// Wsuń/zamknij
bClose_Cmd R= ( (stDigInOut.bI_Closed OR fbTON_CloseTimer.Q) AND NOT bI_SusteinClosePos) OR NOT bI_Control_Ready;
//bClose_Cmd R= ( (bI_Closed OR (fbTON_CloseTimer.Q AND FALSE)) AND NOT bI_SusteinClosePos) OR NOT bI_Control_Ready;
stDigInOut.bQ_Close := bClose_Cmd AND (SEL(bI_MANUAL_CMD, NOT bI_CloseInterlock, NOT (bI_CloseInterlock AND bI_RespectInterlockInMAN)) OR bQ_Closed);
stDigInOut.bQ_Open R= stDigInOut.bQ_Close;

// Wysuń/otwórz
bOpen_Cmd R= ( (stDigInOut.bI_Opened OR fbTON_OpenTimer.Q) AND NOT bI_SusteinOpenPos) OR NOT bI_Control_Ready;
//bOpen_Cmd R= ( (bI_Opened OR (fbTON_OpenTimer.Q AND FALSE)) AND NOT bI_SusteinOpenPos) OR NOT bI_Control_Ready;
stDigInOut.bQ_Open := bOpen_Cmd AND (SEL(bI_MANUAL_CMD, NOT bI_OpenInterlock, NOT (bI_OpenInterlock AND bI_RespectInterlockInMAN)) OR bQ_Opened);
stDigInOut.bQ_Close R= stDigInOut.bQ_Open;

// Określenie sygnałów zamknięcia/otwarcia
fbFTrig_Opened (CLK := stDigInOut.bI_Opened);
fbFTrig_Closed (CLK := stDigInOut.bI_Closed);
IF bAllowOverCrossPosition THEN
	bQ_Opened R= (NOT stDigInOut.bQ_Open AND fbFTrig_Opened.Q) OR stDigInOut.bI_Closed; 
	bQ_Closed R= (NOT stDigInOut.bQ_Close AND fbFTrig_Closed.Q) OR stDigInOut.bI_Opened;
	bQ_Opened S= stDigInOut.bI_Opened;
	bQ_Closed S= stDigInOut.bI_Closed;
ELSE
	bQ_Opened := stDigInOut.bI_Opened;
	bQ_Closed := stDigInOut.bI_Closed; 
END_IF
bCmdActive := FALSE;

// Kontrola czasu pracy siłownika
IF fbTON_OpenTimer.IN AND NOT (stDigInOut.bQ_Open AND NOT bQ_Opened) AND NOT fbTON_OpenTimer.Q THEN
	fMeanFilter(rInputValue := TIME_TO_REAL(fbTON_OpenTimer.ET), rDelta := 10.0, rMeanValue := rOpenMeanTime);
END_IF
fbTON_OpenTimer(IN := stDigInOut.bQ_Open AND NOT bQ_Opened, PT:= REAL_TO_TIME(1000.0*rI_OpenTime));

IF fbTON_CloseTimer.IN AND NOT (stDigInOut.bQ_Close AND NOT bQ_Closed) AND NOT fbTON_CloseTimer.Q THEN
	fMeanFilter(rInputValue := TIME_TO_REAL(fbTON_CloseTimer.ET), rDelta := 10.0, rMeanValue := rCloseMeanTime);
END_IF
fbTON_CloseTimer(IN := stDigInOut.bQ_Close AND NOT bQ_Closed, PT:= REAL_TO_TIME(1000.0*rI_CloseTime));

bInMovement:= fbTON_OpenTimer.IN OR fbTON_CloseTimer.IN;

// Kontrola błędów w pracy
fbTON_controlReady(IN:= bI_Control_Ready, PT:= T#5S);		// Alarmuj tylko po powrocie sygnału gotowości napędów

// Błąd osiągnięcia pozycji otwórz w odpowiednim czasie
IF fbTON_OpenTimer.Q AND fbTON_controlReady.Q AND __ISVALIDREF(fbAlarmTab) THEN
	IF NOT bOpenTimeExceedAlSend THEN
		fbAlarmTab.mPushRow(nAlarmClass:= enAlarmClasses.Error, sMachineId := sActuatorId, sEventDesc := 'Open time exceeded, open position not achieved', dwErrorId := 0);
		bOpenTimeExceedAlSend := TRUE;
	END_IF
ELSE
	bOpenTimeExceedAlSend := FALSE;
END_IF

// Błąd osiągnięcia pozycji zamknij w odpowiednim czasie
IF fbTON_CloseTimer.Q AND fbTON_controlReady.Q AND __ISVALIDREF(fbAlarmTab) THEN
	IF NOT bCloseTimeExceedAlSend THEN
		fbAlarmTab.mPushRow(nAlarmClass:= enAlarmClasses.Error, sMachineId := sActuatorId, sEventDesc := 'Close time exceeded, close position not achieved', dwErrorId := 0);
		bCloseTimeExceedAlSend := TRUE;
	END_IF
ELSE
	bCloseTimeExceedAlSend := FALSE;
END_IF

// Utracenie pozycji otwarcia
fbFTRIG_OpenPosition(CLK:= bQ_Opened);
IF fbFTRIG_OpenPosition.Q AND NOT stDigInOut.bQ_Open AND NOT stDigInOut.bQ_Close AND fbTON_controlReady.Q AND bEnPossLossAlarm AND __ISVALIDREF(fbAlarmTab) THEN
	fbAlarmTab.mPushRow(nAlarmClass:= enAlarmClasses.Error, sMachineId := sActuatorId, sEventDesc := 'Loss open position', dwErrorId := 0);
END_IF

// Utracenie pozycji zamknięcia
fbFTRIG_ClosePosition(CLK:= bQ_Closed);
IF fbFTRIG_ClosePosition.Q AND NOT stDigInOut.bQ_Open AND NOT stDigInOut.bQ_Close AND fbTON_controlReady.Q AND bEnPossLossAlarm AND __ISVALIDREF(fbAlarmTab) THEN
	fbAlarmTab.mPushRow(nAlarmClass:= enAlarmClasses.Error, sMachineId := sActuatorId, sEventDesc := 'Loss close position', dwErrorId := 0);
END_IF

// Kontrola pracy krańcówek
fbRTrig_Open(CLK := stDigInOut.bI_Opened);
fbRTrig_Close(CLK := stDigInOut.bI_Closed);

IF ((stDigInOut.bQ_Open AND fbRTrig_Close.Q AND NOT bAllowOverCrossPosition) OR (stDigInOut.bQ_Close AND fbRTrig_Open.Q AND NOT bAllowOverCrossPosition) OR (stDigInOut.bI_Opened AND stDigInOut.bI_Closed) AND fbTON_controlReady.Q ) AND __ISVALIDREF(fbAlarmTab) THEN
	IF NOT bSwitchesErrorAlSend THEN
		fbAlarmTab.mPushRow(nAlarmClass:= enAlarmClasses.Error, sMachineId := sActuatorId, sEventDesc := 'End stops error', dwErrorId := 0);
	END_IF
ELSE
	bSwitchesErrorAlSend := FALSE;
END_IF

// Ilość cykli pracy
fbRTrig_Ctr_Open (CLK := stDigInOut.bQ_Open);
fbRTrig_Ctr_Close (CLK := stDigInOut.bQ_Close);
IF fbRTrig_Ctr_Open.Q OR fbRTrig_Ctr_Close.Q THEN
	diNbOfOperations := diNbOfOperations+1;
END_IF

ACTION ACT_Stop:
stDigInOut.bQ_Open := stDigInOut.bQ_Close := FALSE;
END_ACTION

METHOD mClose : BOOL
VAR_INPUT
	bManCtrl:BOOL;
END_VAR
IF bManCtrl THEN
	bClose_Cmd S= bI_MANUAL_CMD;
ELSE
	bClose_Cmd S= NOT bI_MANUAL_CMD;
END_IF
bOpen_Cmd R= bClose_Cmd;
bCmdActive := TRUE;
(*bResult := bClose_Cmd;
IF bManCtrl THEN
	bClose_Cmd S= bI_MANUAL_CMD AND NOT (bI_CloseInterlock AND bI_RespectInterlockInMAN);
ELSE
	bClose_Cmd S= NOT bI_MANUAL_CMD AND NOT bI_CloseInterlock;
END_IF
*)
END_METHOD

METHOD mOpen : BOOL
VAR_INPUT
	bManCtrl:BOOL;
END_VAR
IF bManCtrl THEN
	bOpen_Cmd := bI_MANUAL_CMD;
ELSE
	bOpen_Cmd := NOT bI_MANUAL_CMD;
END_IF
bClose_Cmd R= bOpen_Cmd;
bCmdActive := TRUE;
//bResult := bClose_Cmd;
END_METHOD

METHOD mReset : BOOL
VAR_INPUT
END_VAR
// Reset błędów 
fbTON_OpenTimer(IN:= FALSE);
fbTON_CloseTimer(IN:= FALSE);
END_METHOD

METHOD mStop : BOOL
VAR_INPUT
	bManCtrl:BOOL;
END_VAR
IF bManCtrl AND bI_MANUAL_CMD THEN
	bOpen_Cmd := bClose_Cmd := FALSE;
	ACT_Stop();
END_IF
bCmdActive := TRUE;
END_METHOD

END_FUNCTION_BLOCK

// Common/Actuator/fbActuatorV2
FUNCTION_BLOCK fbActuatorV2
VAR_IN_OUT
	
END_VAR
VAR_INPUT
	bControl_Rdy			:BOOL;		// Sygnał gotowości sterowania, sygnały otwórz/zamknij ustawiane tylko gdy jest gotowość
	bInterlock_Open			:BOOL;		// Sygnał blokady otwierania zaworu/napędu (kolizja z innymi elementami)
	bInterlock_Close		:BOOL;		// Sygnał blokady zamykania zaworu/napędu (kolizja z innymi elementami)
	bSusteinOutput			:BOOL;		// Po dojściu do pozycji zadanej podtrzymaj sygnał sterujący - stosować np. dla zaworów 5/2 w celu podtrzymania położenia
	bAllowOvercrossingPos	:BOOL;		// Ustawiaj sygnał otwórz/zamknij gdy ustawi się odpowiednia krańcówka oraz gdy aktywny sygnał sterujący (zejście z krańcówki przy podtrzymaniu nie powoduje zaniku sygnału otwarcia/zamknięcia)
	rOpenTime				:REAL;		//
	rCloseTime				:REAL;
END_VAR
VAR
	stInOuts: stActuatorInOuts;
	fbTON_AllowToNextOper	:TON;
	fbFTrig_Opened: F_TRIG;
	fbFTrig_Closed: F_TRIG;	
	bOpenPos_Overcrossed: BOOL;
	bClosePos_Overcrossed: BOOL;
	fbRTrig_Ctr_OPEN, fbRTrig_Ctr_CLOSE: R_TRIG;
	fbTON_ResetSustein: TON;
END_VAR

VAR PERSISTENT
	udiNbOfOperations:UDINT;
END_VAR

// Reset sygnałów sterujących po osiągnięciu pozycji
fbTON_ResetSustein(IN:= (stInOuts.bQ_Open AND Opened AND NOT bSusteinOutput) OR (stInOuts.bQ_Close AND Closed AND NOT bSusteinOutput),PT:= T#250MS);
stInOuts.bQ_Open R= stInOuts.bQ_Open AND ( (bInterlock_Open AND NOT Opened) OR fbTON_ResetSustein.Q);
stInOuts.bQ_Close R= stInOuts.bQ_Close AND ( (bInterlock_Close AND NOT Closed) OR fbTON_ResetSustein.Q);

// Zezwolenie na kolejną operację nie szybciej niż co 50 ms
fbTON_AllowToNextOper(IN:= NOT stInOuts.bQ_Open AND NOT stInOuts.bQ_Close, PT:= T#50MS);

// Określenie sygnałów zamknięcia/otwarcia
fbFTrig_Opened (CLK := stInOuts.bI_Opened);
fbFTrig_Closed (CLK := stInOuts.bI_Closed);
bOpenPos_Overcrossed S= stInOuts.bQ_Open AND fbFTrig_Opened.Q;
bOpenPos_Overcrossed R= stInOuts.bQ_Close AND fbFTrig_Opened.Q;
bClosePos_Overcrossed S= stInOuts.bQ_Close AND fbFTrig_Closed.Q;
bClosePos_Overcrossed R= stInOuts.bQ_Open AND fbFTrig_Closed.Q;

// Ilość cykli pracy
fbRTrig_Ctr_OPEN (CLK := stInOuts.bQ_Open);
fbRTrig_Ctr_CLOSE (CLK := stInOuts.bQ_Close);
IF fbRTrig_Ctr_OPEN.Q OR fbRTrig_Ctr_CLOSE.Q THEN
	udiNbOfOperations := udiNbOfOperations+1;
END_IF

METHOD mClose : BOOL
IF Closed THEN		// Siłownik zamknięty spróbuj ustawić wyjście		
	stInOuts.bQ_Open := FALSE;
	stInOuts.bQ_Close S= bControl_Rdy AND bSusteinOutput; 
	mClose := TRUE;
ELSE	// Jeśli siłownik nie zamknięty spróbuj ustawić wyjscie
	stInOuts.bQ_Close S= stInOuts.bQ_Open R= NOT bInterlock_Close AND bControl_Rdy;
END_IF
END_METHOD

METHOD mOpen : BOOL
IF Opened THEN			// Siłownik otwarty spróbuj ustawić wyjście	
	stInOuts.bQ_Close := FALSE;
	stInOuts.bQ_Open S= bControl_Rdy AND bSusteinOutput; 
	mOpen := TRUE;
ELSE					// Jeśli siłownik nie zamknięty spróbuj ustawić wyjscie
	stInOuts.bQ_Open S= stInOuts.bQ_Close R= NOT bInterlock_Open AND bControl_Rdy;
END_IF
END_METHOD

METHOD mReset : BOOL
END_METHOD

METHOD mStop : BOOL
stInOuts.bQ_Open := stInOuts.bQ_Close := FALSE;
END_METHOD

PROPERTY Closed : BOOL
GET
Closed := stInOuts.bI_Closed OR (bAllowOvercrossingPos AND bClosePos_Overcrossed);
END_GET
END_PROPERTY

PROPERTY CmdsCounter : UDINT
GET
CmdsCounter := udiNbOfOperations;
END_GET
SET
udiNbOfOperations := CmdsCounter;
END_SET
END_PROPERTY

PROPERTY Moving : BOOL
GET
Moving := (stInOuts.bQ_Open AND NOT Opened)OR (stInOuts.bQ_Close AND NOT Closed);
END_GET
END_PROPERTY

PROPERTY Opened : BOOL
GET
Opened := stInOuts.bI_Opened OR (bAllowOvercrossingPos AND bOpenPos_Overcrossed);
END_GET
END_PROPERTY

END_FUNCTION_BLOCK

// Common/AlarmTable/f_AlarmClassToUINT
FUNCTION f_AlarmClassToUINT : UINT
VAR_INPUT
	nAlarmType:enAlarmClasses;
END_VAR
VAR
END_VAR

CASE nAlarmType OF
	enAlarmClasses.None, enAlarmClasses.Info:
		f_AlarmClassToUINT:= 1;
	enAlarmClasses.Warning:
		f_AlarmClassToUINT:= 2;
	enAlarmClasses.Error:
		f_AlarmClassToUINT:= 3;
	enAlarmClasses.Quality:
		f_AlarmClassToUINT:= 4;
	enAlarmClasses.Maintenance:
		f_AlarmClassToUINT:= 5;
	enAlarmClasses.IT:
		f_AlarmClassToUINT:= 6;
	enAlarmClasses.Developer:
		f_AlarmClassToUINT:= 7;
END_CASE

END_FUNCTION

// Common/AlarmTable/f_AlarmEnableTest
FUNCTION f_AlarmEnableTest : BOOL
VAR_INPUT
	uiLogSettings:UINT;
	nAlarmType:enAlarmClasses;
END_VAR
VAR
	iBase:UINT := 1;
	uiBitNb: UINT;
END_VAR

CASE nAlarmType OF
	enAlarmClasses.None:
		f_AlarmEnableTest := FALSE;
		RETURN;	
	enAlarmClasses.Info:
		uiBitNb:= 0;
	enAlarmClasses.Warning:
		uiBitNb:= 1;
	enAlarmClasses.Error:
		uiBitNb:= 2;
	enAlarmClasses.Quality:
		uiBitNb:= 3;
	enAlarmClasses.Maintenance:
		uiBitNb:= 4;
	enAlarmClasses.IT:
		uiBitNb:= 5;
	enAlarmClasses.Developer:
		uiBitNb:= 6;
END_CASE
f_AlarmEnableTest := (ROL(iBase,uiBitNb) AND uiLogSettings) > 0;

END_FUNCTION

// Common/AlarmTable/fbAlarmMasterTable
FUNCTION_BLOCK PUBLIC fbAlarmMasterTable
VAR CONSTANT
	uiMaxRows:UINT := 200;	// nie powinno być mniejsze niż 50, nie może być mniejsze niż 25!
END_VAR
VAR_OUTPUT
	astErrTable: ARRAY [1..uiMaxRows] OF stAlarmTableRow;		// Tabela z błędami
	uiRowNumber:UINT;		// Aktualna liczba wierszy w tabeli
END_VAR

METHOD mPopRows : BOOL
VAR_IN_OUT
	fbSimpleAlarm:fbAlarmSlaveTable;
END_VAR

IF fbSimpleAlarm.uiRowsToRead > 0 AND fbSimpleAlarm.uiRowsToRead <= 20 THEN
	// Przesuń obecne alarmy
	MEMMOVE (srcAddr := ADR(astErrTable[1]), destAddr := ADR(astErrTable[1+fbSimpleAlarm.uiRowsToRead]), n := (MIN((uiMaxRows-fbSimpleAlarm.uiRowsToRead), uiRowNumber)*SIZEOF(astErrTable[1])) );
	// Gdy obecne alarmy przesunięte dodaj nowe
	MEMMOVE (srcAddr := ADR(fbSimpleAlarm.astErrTable[1]), destAddr := ADR(astErrTable[1]), n := (fbSimpleAlarm.uiRowsToRead*SIZEOF(astErrTable[1])) );
	uiRowNumber := LIMIT(0,uiRowNumber + fbSimpleAlarm.uiRowsToRead,uiMaxRows);
	fbSimpleAlarm.aMesagesPoped();
END_IF
END_METHOD

METHOD mPushRow : BOOL
VAR_INPUT
	nAlarmClass:enAlarmClasses :=enAlarmClasses.Info;
	sMachineId:STRING(30);
	sEventDesc:STRING;
	dwErrorId:DWORD;
END_VAR
// Dodaj nowy alarm tylko gdy inny niż ostatni, jeśli taki sam zaktualizuj czas wystąpienia oraz zwiększ licznik wystąpień
IF sMachineId = astErrTable[1].sMachineId AND sEventDesc = astErrTable[1].sEventDescription THEN
	astErrTable[1].dtEventTime:= GVL_Aircom.stAC_DT_Data.dtActualDate;
	astErrTable[1].uiRepeatQty:= astErrTable[1].uiRepeatQty +1;
ELSE
	MEMMOVE (srcAddr := ADR(astErrTable[1]), destAddr := ADR(astErrTable[2]), n := ((uiMaxRows-1)*SIZEOF(astErrTable[1])) );
	astErrTable[1].dtEventTime:= GVL_Aircom.stAC_DT_Data.dtActualDate;
	astErrTable[1].sMachineId := sMachineId;
	astErrTable[1].sEventDescription := sEventDesc;
	astErrTable[1].dwErrorCode := dwErrorId;
	astErrTable[1].nAlarmClass := nAlarmClass;
	astErrTable[1].uiRepeatQty := 0;
	uiRowNumber := LIMIT(0,uiRowNumber +1,uiMaxRows);
END_IF
END_METHOD

METHOD mReset : BOOL
VAR_INPUT
END_VAR

VAR
END_VAR
MEMSET(destAddr := ADR(astErrTable), fillByte := 0, n := SIZEOF(astErrTable)); 
uiRowNumber := 0;
END_METHOD

END_FUNCTION_BLOCK

// Common/LoadCell/fLoadCellCtrl
FUNCTION fLoadCellCtrl : WORD
VAR_INPUT
	bStartCalibration: BOOL;		
	bDisableCalibration:BOOL;
	bInputFreeze:BOOL;	
	bTara:BOOL;	
END_VAR
VAR	
END_VAR

fLoadCellCtrl := 0;
fLoadCellCtrl.0 := bStartCalibration;
fLoadCellCtrl.1 := bDisableCalibration;
fLoadCellCtrl.2 := bInputFreeze;
fLoadCellCtrl.4 := bTara;

END_FUNCTION

// Common/LoadCell/fLoadCellStatusToBOOL
FUNCTION fLoadCellStatusToBOOL : BOOL
VAR_INPUT
	wStatus:	WORD;	// Measurement status from Module
END_VAR
VAR
	bError: BOOL;		// Błąd pomiaru
	bOverrange:BOOL;
	bDataInvalud:BOOL;	
	bCalInProgress:BOOL;	
	bSteadyState:BOOL;	
	SyncErr:BOOL;	
	bTxPDO_Toggle:BOOL;	//	Toogle gdy jest nowa wartość 
END_VAR

bOverrange := wStatus.1;
bDataInvalud := wStatus.3;
bError := wStatus.6;
bCalInProgress := wStatus.7;
bSteadyState := wStatus.8;
SyncErr := wStatus.13;
bTxPDO_Toggle := wStatus.15;

END_FUNCTION

// Common/Maintenance/fbIIS_Restart
FUNCTION_BLOCK PUBLIC fbIIS_Restart
VAR_INPUT
	bExecute:BOOL;
END_VAR
VAR_OUTPUT
	bBusy:BOOL;
	bError:BOOL;
	ErrID: UDINT;
END_VAR
VAR
	NT_StartCMD:NT_StartProcess;
END_VAR

NT_StartCMD(
	NETID:= '', 
	PATHSTR := 'C:\TwinCAT\AC_Reset_Services\ResetIIS.bat',
	DIRNAME := 'C:\TwinCAT\AC_Reset_Services',
	COMNDLINE:= '', 
	START:= bExecute, 
	TMOUT:= T#15S, 
	BUSY=> bBusy, 
	ERR=> , 
	ERRID=> );
IF NT_StartCMD.ERR THEN
	bError := TRUE;
	ErrID:= NT_StartCMD.ERRID;
END_IF

END_FUNCTION_BLOCK

// Common/Maintenance/fbTcAdsWcfHost_Restart
FUNCTION_BLOCK PUBLIC fbTcAdsWcfHost_Restart
VAR_INPUT
	bExecute:BOOL;
END_VAR
VAR_OUTPUT
	bBusy:BOOL;
	bError:BOOL;
	ErrID: UDINT;
END_VAR
VAR
	NT_StartCMD:NT_StartProcess;
	fbTON_Reset:TON;
	fbRTRIG_Start: R_TRIG;
END_VAR

fbRTRIG_Start(CLK:= bExecute);		
IF fbRTRIG_Start.Q THEN
	bError:= FALSE;
	bBusy:= TRUE;
	NT_StartCMD(START := FALSE);
END_IF
IF bBusy THEN
	NT_StartCMD(
		PATHSTR := 'C:\TwinCAT\AC_Reset_Services\ResetTcAdsWcfHost.bat',
		DIRNAME := 'C:\TwinCAT\AC_Reset_Services',
		COMNDLINE:= '', 
		START:= fbRTRIG_Start.Q, 
		TMOUT:= T#10S);
	
	IF NT_StartCMD.ERR THEN
		bError := TRUE;
		bBusy := FALSE;
		ErrID:= NT_StartCMD.ERRID;
	ELSIF NOT NT_StartCMD.BUSY THEN
		bError := FALSE;
		bBusy := FALSE;
	END_IF
END_IF
fbTON_Reset(IN:= bBusy, PT:= T#5s);
IF fbTON_Reset.Q THEN
	bError:= TRUE;
	bBusy:= FALSE;
END_IF

END_FUNCTION_BLOCK

// Common/Measurement_Analog/fACRoundReal
FUNCTION fACRoundReal : REAL
VAR_INPUT
	rIn:REAL;
	iFracDigits:INT;
END_VAR
VAR
	rScaler: REAL;
	diScaledValue:DINT;
END_VAR

iFracDigits := LIMIT(1,iFracDigits,6);
rScaler:= EXPT(10,iFracDigits);
diScaledValue := REAL_TO_DINT(rScaler*rIn+ SEL(FRAC(rScaler*rIn)<5,1,0));
fACRoundReal:= DINT_TO_REAL(diScaledValue)/rScaler;

END_FUNCTION

// Common/Measurement_Analog/FB_FilterEx
//==================================================================================================
//							Beckhoff Automation Poland
//									23.11.2016
//			Bloczek do filtru inercyjnego do wygladzania przebiegow,					
//					czas próbkowania wyliczany wewnętrznie
//  v1.1	|| TC v 3.1.4020.28		|| - poprawienie inicjaLLzacji, notacja wegierska
// 	v1.0	|| TC v 3.1.4020.0		|| - pierwsza wersja
//==================================================================================================
FUNCTION_BLOCK FB_FilterEx
VAR_INPUT
	rIn										: REAL;					// Sygnal wejsciowy
	tTimeConstant							: TIME;					// Stala czasowa T gdy rOut = 0,63 * rIn 
END_VAR
VAR_OUTPUT
	rOut									: REAL;					// Przefiltrowany sygnal wyjsciowy, 
END_VAR
VAR
	rLastOut								: REAL;					// Wartosc wyjscia w poprzednim cyklu
	rCycleTime								: REAL; 				// [ms]
	rTimeConst								: REAL;					// [ms]
	tX										: TIME;					// Aktualny czas
	tY 										: TIME;					// Zmienna pomocnicza, poprzedni czas
	tCycleTime								: TIME;					// Wyliczony czas cyklu
	bFirstCycle								: BOOL := TRUE;			// Flaga pierwszego cyklu - nie mamy jeszce wyliczonego prawidlowo czasu cylu 
																	// - potrzebujemy dwoch cylki do odjecia czasu
END_VAR

// Obliczenie czasu cyklu do inkrementu
tX 					:= TIME();
IF NOT bFirstCycle THEN
	tCycleTime 		:= tX - tY;
END_IF
tY 					:= tX;
// Przeliczenie czasu na typ REAL
rCycleTime 			:= TIME_TO_REAL(tCycleTime);
rTimeConst 			:= TIME_TO_REAL(tTimeConstant);
// Wyliczenie wyjscia tylko jesli stala czasowa wieksza od 1 ms i zakonczylismy inicjaLLzacje
IF NOT bFirstCycle AND rTimeConst > 0.001 THEN
	rOut 			:= rLastOut + (rIn - rLastOut) * rCycleTime/rTimeConst;
	rLastOut 		:= rOut;
END_IF
// Zerowanie flagu pierwszego cyklu
bFirstCycle 		:= FALSE;

END_FUNCTION_BLOCK

// Common/Measurement_Analog/fbAnalogMeasurement
FUNCTION_BLOCK fbAnalogMeasurement
VAR_INPUT
	rIn:REAL;				// Wejście pomiarowe
	bExtError:BOOL;			// Sygnał zewnętrzebgo błędu
	stMeasureScalingData:stMeasurementScalingData;		// Dane do skalowania
	tStalaCzasowa:TIME;
END_VAR
VAR_OUTPUT
	rOutFiltered:REAL;
	bMeasurementOK:BOOL;
END_VAR
VAR
	fbFiltr_1 : FB_FilterEx;
	rRange_RAW: REAL;
	rRange_ENG: REAL;
	rMeasurement: REAL;
	rErrorLimit: REAL;
END_VAR

rRange_RAW := stMeasureScalingData.rScalingRawValue_II - stMeasureScalingData.rScalingRawValue_I;
rRange_ENG := stMeasureScalingData.rScalingEngValue_II - stMeasureScalingData.rScalingEngValue_I;
rErrorLimit := 0.05* rRange_ENG;

IF ABS(rRange_RAW) > 0.0001 THEN
	rMeasurement:= ( (rIn - stMeasureScalingData.rScalingRawValue_I)/rRange_RAW )*rRange_ENG + stMeasureScalingData.rScalingEngValue_I;
END_IF

bMeasurementOK := NOT bExtError AND (rMeasurement > (stMeasureScalingData.rScalingEngValue_II - rErrorLimit) AND rMeasurement < (stMeasureScalingData.rScalingEngValue_I + rErrorLimit) );

fbFiltr_1(rIn := rMeasurement, tTimeConstant := tStalaCzasowa, rOut => rOutFiltered);

END_FUNCTION_BLOCK

// Common/Measurement_Analog/fbAnalogMonitor
FUNCTION_BLOCK fbAnalogMonitor
VAR_INPUT
	rIN			: REAL; 	// Input value
	tTactTime	: TIME;		// Time periot between collecting samples
END_VAR
VAR_OUTPUT
	rMeanValue	: REAL;
	bStable		: BOOL;
	bRising		: BOOL;
	bFalling	: BOOL;
	bTrendChangeRising	: BOOL;
	bTrendChangeFalling	: BOOL;
END_VAR
VAR
	arValues	: ARRAY [1..10] OF REAL;	//
	fbTON_Tact	: TON;
	rSumOfValuesInArray, rDivider: REAL;
	rMean12, rMean56, rMean910: REAL;
	rStableFactor: REAL;
END_VAR

fbTON_Tact(IN:= NOT fbTON_Tact.Q,PT:= tTactTime);

IF fbTON_Tact.Q THEN
	fbTON_Tact(IN:= FALSE);
	rSumOfValuesInArray := rSumOfValuesInArray - arValues[10];
	rDivider := LIMIT(1,rDivider+1,10);  
	MEMMOVE(srcAddr := ADR(arValues[1]), destAddr := ADR(arValues[2]),n:= 36);
	arValues[1] := rIN;
	rSumOfValuesInArray := rSumOfValuesInArray + arValues[1];
	rMeanValue := rSumOfValuesInArray/rDivider;
	rMean12 := (arValues[1]+ arValues[2])/2.0; 
	rMean56 := (arValues[5]+ arValues[6])/2.0;
	rMean910 := (arValues[9]+ arValues[10])/2.0; 
	bStable := bRising := bFalling := bTrendChangeRising := bTrendChangeFalling := FALSE;
	rStableFactor:= 0.1*rMeanValue;
	IF ABS(rMean12-rMeanValue)< rStableFactor AND ABS(rMean56-rMeanValue)< rStableFactor AND ABS(rMean910-rMeanValue)< rStableFactor THEN
		bStable := TRUE;
	ELSIF rMean12 > rMean56 AND rMean56 > rMean910 THEN
		bRising := TRUE;
	ELSIF rMean910 > rMean56 AND rMean56 > rMean12 THEN
		bFalling := TRUE;
	ELSIF rMean910 > rMean56 AND rMean56 < rMean12 THEN
		bTrendChangeRising := TRUE;
	ELSIF rMean910 < rMean56 AND rMean56 > rMean12 THEN
		bTrendChangeFalling := TRUE;
	END_IF
END_IF

END_FUNCTION_BLOCK

// Common/Measurement_Analog/fMeasureStatusToBOOL
// Funkcja rozbija status na pojedyncze zmeinne - przy wywołaniu zwracana wartość BOOL równa się aktywnemu błędowi
FUNCTION fMeasureStatusToBOOL : BOOL
VAR_INPUT
	wStatus:	WORD;	// Measurement status from Module
END_VAR
VAR_OUTPUT
	bError: BOOL;		// Błąd pomiaru
	bUnderrange:BOOL;
	bOverrange:BOOL;
	bLim1_LessEq:BOOL;	//	Wartość mniejsza/równa Limit1
	bLim1_GreatEq:BOOL;	//	Wartość większa/równa Limit1
	bLim2_LessEq:BOOL;	//	Wartość mniejsza/równa Limit2
	bLim2_GreatEq:BOOL;	//	Wartość większa/równa Limit2
	bTxPDO_State:BOOL;	// 
	bTxPDO_Toggle:BOOL;	//	Toogle gdy jest nowa wartość 
END_VAR

bUnderrange := wStatus.0;
bOverrange := wStatus.1;
bLim1_LessEq := wStatus.2;
bLim1_GreatEq := wStatus.3;
bLim2_LessEq := wStatus.4;
bLim2_GreatEq := wStatus.5;
fMeasureStatusToBOOL := bError := wStatus.6;
bTxPDO_State := wStatus.14;
bTxPDO_Toggle := wStatus.15;

END_FUNCTION

// Common/Measurement_Analog/fRealValueFilter
FUNCTION fRealValueFilter : REAL
VAR_INPUT
	rIn:REAL;
	rDelta:REAL;
	bSquaredE:BOOL;	
END_VAR
VAR_IN_OUT
	rMeanValue:REAL;
END_VAR
VAR
	rE: REAL;
END_VAR

rDelta := LIMIT(1,rDelta,100);
IF ABS(0.20*rMeanValue) < ABS( (rMeanValue - rIn)/rDelta) THEN	// Wpisanie aktualnej wartości przy starcie
	rMeanValue := rIn;
END_IF
rE:= (rMeanValue - rIn);
IF bSquaredE THEN
	rMeanValue := rMeanValue - (ABS(rE)*rE)/rDelta;	
ELSE
	rMeanValue := rMeanValue - rE/rDelta; 	
END_IF

END_FUNCTION

// Common/PulseCounter/fbPulseCounter
FUNCTION_BLOCK PUBLIC fbPulseCounter
VAR_INPUT
	bImpulseSignal:BOOL;
	rValuePerImpulse:REAL;
	rNewCounterValue:REAL;
	bSaveNewValue:BOOL;
END_VAR
VAR_OUTPUT
	rCounterValue:REAL;
END_VAR
VAR 
	fbTON_ContactVibrFilter:TON;
	fbRTRIG_ImpulseON:R_TRIG;
	fbRTRIG_MoveNewValue:R_TRIG;
	rCounterMemLastShift:REAL;
	rUsageMemLastShift:REAL;
	bStartUp:BOOL:=TRUE;
END_VAR
VAR PERSISTENT
	rCounterValuePersistant:REAL;
	liImpulseCounter:LINT;
END_VAR

fbTON_ContactVibrFilter(IN := bImpulseSignal, PT:= T#25MS);
fbRTRIG_ImpulseON(CLK:= fbTON_ContactVibrFilter.Q); 
fbRTRIG_MoveNewValue(CLK:= bSaveNewValue);

IF bStartUp THEN
	rCounterValue := rCounterValuePersistant;
	bStartUp := FALSE;
END_IF
IF fbRTRIG_MoveNewValue.Q THEN
	rCounterValuePersistant := rNewCounterValue;
END_IF

IF fbRTRIG_ImpulseON.Q THEN
	liImpulseCounter := liImpulseCounter +1;
	rCounterValuePersistant := rCounterValuePersistant + rValuePerImpulse;
	rCounterValue := rCounterValuePersistant;
END_IF

END_FUNCTION_BLOCK

// Common/PulseCounter/fbPulseCounterPIM
FUNCTION_BLOCK PUBLIC FINAL fbPulseCounterPIM EXTENDS fbPulseCounter
VAR_INPUT
	I_Sql: I_SqlCmds;
	bSaveCtr: BOOL;
	bCtrType_0Elec_1Air: BOOL;
END_VAR
VAR_OUTPUT
END_VAR
VAR	
	fbRTRIG_Save:R_TRIG;
	iCallsCtr_OK, iCallsCtr_ERR:INT;
	tOffset: TIME;
	fbTON_Delay: TON;
	bResult: BOOL;
END_VAR

SUPER^();
IF GVL_Aircom.bInit OR tOffset = T#0S THEN
	GVL_Aircom.fbRand(Seed:= TIME_TO_INT(GVL_Aircom.stAC_DT_Data.tActualTime));
	tOffset := LREAL_TO_TIME(GVL_Aircom.fbRand.Num*30000.0);
END_IF
IF I_Sql <> 0 THEN
	fbRTRIG_Save(CLK:= bSaveCtr);
	fbTON_Delay.IN S= fbRTRIG_Save.Q; 
	fbTON_Delay(PT:= tOffset);
	IF fbTON_Delay.Q THEN
		IF bCtrType_0Elec_1Air THEN
			bResult:= I_Sql.m_SqlInsCompressedAirConsumption(rActCompressedAirConsumption := rCounterValue);
		ELSE
			bResult:= I_Sql.m_SqlInsEnergyConsumption(rActEnergyConsumption := rCounterValue);
		END_IF
		IF bResult THEN	iCallsCtr_OK := iCallsCtr_OK + 1;
		ELSE iCallsCtr_ERR := iCallsCtr_ERR + 1;
		END_IF
		fbTON_Delay.IN:= FALSE;
	END_IF
END_IF

END_FUNCTION_BLOCK

// PIM/Interfaces/I_SqlCmds
INTERFACE I_SqlCmds

// Zapis do DB dodatkowego kodu błędu - jeśli rozkaz dodany do kolejki zmienna wyjściowa ma wartość TRUE, jeśli nie (błąd dodania) FALSE
METHOD m_SqlInsAdditionalError : BOOL
VAR_INPUT
	sErrCode:STRING(10);		// Kod błędu do wysłania
END_VAR
END_METHOD

// Zapis do DB licznika zużycia powietrza - jeśli rozkaz dodany do kolejki zwraca TRUE, jeśli nie FALSE
METHOD m_SqlInsCompressedAirConsumption : BOOL
VAR_INPUT
	rActCompressedAirConsumption:REAL;		// Wartość licznika zużycia sprężonego powietrza
END_VAR
END_METHOD

// Zapis do DB relacji ostatniego statusu z kodem błędu - jeśli rozkaz dodany do kolejki zwraca TRUE, jeśli nie FALSE
METHOD m_SqlInsDefectRelation : BOOL
VAR_INPUT
	sErrCode:STRING(10);			// Kod błędu
END_VAR
END_METHOD

// Zapis do DB licznika zużycia energi na stanowisku - jeśli rozkaz dodany do kolejki zwraca TRUE, jeśli nie FALSE
METHOD m_SqlInsEnergyConsumption : BOOL
VAR_INPUT
	rActEnergyConsumption:REAL;			// Wartość licznika zużycia energii elektrycznej
END_VAR
END_METHOD

// Zapis do DB danych rozszerzonych operacji - jeśli rozkaz dodany do kolejki zwraca TRUE, jeśli nie FALSE
METHOD m_SqlInsertExtendedData : BOOL		
VAR_INPUT
	pParameters: POINTER TO BYTE;				// Wskaźnik na tablicę elementów typu PIM_ExtDataRow
	uiArraySize: UINT;							// Rozmiar tablicy parametrów (może być pojedyncza zmienna)
END_VAR
END_METHOD

// Zapis do DB statusu ostatniej operacji - gdy rozkaz zostanie wykonany zwraca TRUE
METHOD m_SqlSelInsStatus : BOOL
VAR_INPUT
	bStatus:BOOL:= FALSE;		// Status operacji do zapisania
	sErrCode:STRING(10);		// kod błędu - tylko jeśli status  FALSE
	bSustein:BOOL:= FALSE;		// Jeśli TRUE po wywołaniu przez FbMaszyny wykonwyanie rozkazu przerzucone na fbStation (wysyłanie rozkazu w tle)- ustawiana odpowiednia flaga 
END_VAR
VAR_OUTPUT
	bProcessing:BOOL;			// Przetwarzanie rozkazu trwa (rozkaz dodany do kolejki)
	bResultOK:BOOL;				// Wynik wykonania rozkazu (do sprawdzenia gdy metoda zwróci TRUE)
	liStatusId:LINT;			// Id statusu części w DB
END_VAR
END_METHOD

// Pobranie z DB statusu ostatniej operacji dla danego DM z poprzedniego stanowiska - gdy rozkaz zostanie wykonany zwraca TRUE
METHOD m_SqlSelLastOperationStatus : BOOL
VAR_INPUT
	sCodeDM:STRING(255);		// Identyfikator części (kod DataMatrix)
END_VAR
VAR_OUTPUT
	bProcessing:BOOL;			// Przetwarzanie rozkazu trwa (rozkaz dodany do kolejki)
	bResultOK:BOOL;				// Wynik wykonania rozkazu (do sprawdzenia gdy metoda zwróci TRUE)
	bPrevOperStat:BOOL;			// Status ostatniej operacji na poprzednim stanowisku
END_VAR
END_METHOD

END_INTERFACE

// Common/RecipeManager/fbRecipeManager
FUNCTION_BLOCK fbRecipeManager
VAR CONSTANT
	iMaxRecipeNumber:INT:=40;		// If you change this value, you must also update astRecipeList array size (same value)
	uiMaxStructureSize:UINT:= 1024;
END_VAR
VAR_INPUT
	sRecipesDirectory:STRING;
	pPLC_Struct:POINTER TO BYTE;
	uiPLC_StructSize:UINT;
	pTMP_PLC_Struct:POINTER TO BYTE;				// Struktura pomocnicza - konieczna do deklaracji
	bTextFormat:BOOL:= FALSE;
END_VAR
VAR_OUTPUT
	bError:BOOL;
	nErrorCode:nRecipeManager_ErrorList;
END_VAR
VAR
	fbFileOpen:FB_FileOpen;
	fbFileRead:FB_FileRead;
	fbFileWrite:FB_FileWrite;
	fbFileClose:FB_FileClose;
	fbFileDelete:FB_FileDelete;
	fbReloadRecipes:FB_EnumFindFileEntry;
	
	// HMI variables
	sRecipeName:STRING;
	bReloadRecipes:BOOL;
	bWriteRecipe:BOOL;
	bReadRecipe:BOOL;
	bCopyTMP_2_PLC:BOOL;
	bCopyPLC_2_TMP:BOOL;
	
	
	uiStructSize:UINT;
	bWritingRecipe: BOOL;
	iStep: INT;
	fbTON_StepTimeout: TON;
	hFiileHandler: UINT;
	uiErrorID: UDINT;
	bRecipeSave_OK: BOOL;
	bReadingRecipe: BOOL;
	bRecipeRead_OK: BOOL;
	bPointerValid: BOOL;
	bRefreshRecipeList: BOOL;
	bRecipeList_Reloaded: BOOL;
	bFirstEntry: BOOL;
	bAbort: BOOL;
	astRecipeList:ARRAY [1..40] OF stRecipeManager_ListEntry;
	iNbOfFoundRecipes: INT;
	bRefreshingRecipeList: BOOL;
	bResetInternal: BOOL;
	iTableSelIndex:INT;
	bTableRowSelected:BOOL;
	wCRCsum: WORD;
	bSizeNotEqual: BOOL;
	wCRCsumReaded: WORD;
	bFileOpen: BOOL;
	bCloseFileAfterError: BOOL;
	nErrorCodeMemory:INT;
	iTableSelIndexMemory: INT;
	bSavePLCStruct: BOOL;
	bDeleteRecipe: BOOL;
	bDeletingRecipe: BOOL;
	bRecipeDeleted_OK: BOOL;
	bDeleteConfirmed: BOOL;
	bCopyTMP_2_PLC_Confirmed: BOOL;
	fbRTRIG_ReloadList: R_TRIG;
	fbTON_OKSigReset: TON;
	fbTON_DeleteConfirmWindowReset: TON;
	fbTON_Copy2PLCConfirmWindowReset: TON;
END_VAR

(*
******************************************* Recipe Manager *******************************************

Jako wejście podajemy adres struktury w króre są przechowywane dane (struktury docelowej pPLC_Struct oraz tymczasowej używanej jako bufor panmięci pTMP_PLC_Struct). 

Format zapisu struktury - Dane są zapisywane jako postać binarna - struktura nie powinna zmieniać swojej postaci!. Jeśli koniecznie należy dodać zmienną do struktury
należy dodawać na końcu struktury. Wtedy gdy zapisana receptura nie ma wystarczającej ilości danych, struktura w PLC uzupełniana jest tylko do rozmiaru zawartego w recepturze.
Każda reseptura jest zapisana w poniższym formacie: 
	- pierwsze 2 bajty to rozmiar danych w strukturze (dane są umiejscowione zgodnie z formatem struktury od 3-go bajtu
	- n bajtów danych struktury
	- ostatnie dwa bajty to suma CRC16 obliczana z danych struktury (PRZED ZAPISEM DANYCH STRUKTURY NALEŻY WYZEROWAĆ PAMIĘĆ STRUKTURY aby nieużywane bajty nie wpłyneły na sumę CRC!!!)
	
Współpraca z PIM:
Podczas zalogowania użytkownika sterownik automatycznie odpytuje bazę danych o sumę CRC aktualnej wersji parametrów (trzeba też odczytać parametry urządzenia np zgrzewarki), 
baza danych (DB) zwraca zatwierdzoną aktualną sumę CRC, następuje porównanie sumy CRC z DB oraz z urządzenia. W razie zgodności urządzenie jest dopuszczone do pracy, inaczej jest blokowane

Konfiguracja - w przypadku gdy w DB nie ma parametrów lub parametry w maszynie są nieaktualne trzeba nadpisać aktywny zestaw parametrów w DB.
Istnieje możliwość zapisu aktualnych parametrów do DB, w tym celu system PIM ustawia odpowiednią zmienną, po ustawieniu sterownik PLC pobiera dane z maszyny oraz wysyła do DB wraz z nową sumą CRC

*)

bPointerValid := pTMP_PLC_Struct > 0 AND pPLC_Struct > 0 AND uiPLC_StructSize > 0;

IF (bWriteRecipe OR bWritingRecipe) AND NOT bReadingRecipe AND NOT bRefreshingRecipeList AND bPointerValid AND LEN(sRecipeName) > 2 THEN
	ACT_WriteRecipe();
	bWriteRecipe := FALSE;
	bRecipeList_Reloaded := FALSE;
END_IF

IF (bReadRecipe OR bReadingRecipe) AND NOT bWritingRecipe AND NOT bRefreshingRecipeList AND bPointerValid AND bRecipeList_Reloaded AND bTableRowSelected THEN
	ACT_ReadRecipe();
	bReadRecipe := FALSE;
END_IF

IF (bReloadRecipes OR bRefreshingRecipeList) AND NOT bWritingRecipe AND NOT bReadingRecipe THEN
	ACT_RefreshRecipeList();
	bReloadRecipes := FALSE;
END_IF

IF ((bDeleteRecipe AND bDeleteConfirmed) OR bDeletingRecipe) AND NOT bReadingRecipe AND NOT bRefreshingRecipeList AND NOT bWritingRecipe AND bTableRowSelected THEN
	ACT_DeleteRecipe();
	bDeleteConfirmed := bDeleteRecipe := FALSE;
	bRecipeList_Reloaded := FALSE;
END_IF
fbTON_DeleteConfirmWindowReset(IN:= bDeleteRecipe, PT:= T#15S);
bDeleteRecipe R= fbTON_DeleteConfirmWindowReset.Q;

IF (bWriteRecipe AND NOT bWritingRecipe) OR (bReadRecipe AND NOT bReadingRecipe) OR (bReloadRecipes AND NOT bRefreshingRecipeList) OR (bDeleteConfirmed AND NOT bDeletingRecipe) THEN
	nErrorCode := nRecipeManager_ErrorList.CommandStartProgramError;
	bWriteRecipe := bReadRecipe := bReloadRecipes := bDeleteRecipe := bDeleteConfirmed := FALSE;
END_IF

fbRTRIG_ReloadList(CLK:= (bRecipeDeleted_OK AND NOT bDeletingRecipe) OR (bRecipeSave_OK AND NOT bWritingRecipe));
IF fbRTRIG_ReloadList.Q THEN
	bReloadRecipes:= TRUE;
END_IF

fbTON_OKSigReset(IN:= bRecipeDeleted_OK OR bRecipeRead_OK OR bRecipeSave_OK, PT:= T#5S);
IF fbTON_OKSigReset.Q THEN
	bRecipeDeleted_OK := bRecipeRead_OK := bRecipeSave_OK := FALSE;
END_IF

IF bResetInternal THEN
	iStep := 0;	
	IF bFileOpen THEN
		fbFileClose(bExecute:= FALSE);
		fbFileClose(hFile:= hFiileHandler, 
			bExecute:= TRUE, 
			tTimeout:= T#1S,);
		IF NOT fbFileClose.bBusy THEN
			IF fbFileClose.bError THEN
				uiErrorID:= fbFileClose.nErrId;
				nErrorCodeMemory := nRecipeManager_ErrorList.NoError;
				nErrorCode := nRecipeManager_ErrorList.FileCloseError;
				bResetInternal := FALSE;
			ELSE
				bFileOpen := FALSE;
				bResetInternal := FALSE;
				nErrorCodeMemory := nErrorCode := nRecipeManager_ErrorList.NoError;
				bError := FALSE;
			END_IF
			fbFileClose(bExecute:= FALSE);
		END_IF
	ELSE
		bResetInternal := FALSE;
		nErrorCodeMemory := nErrorCode := nRecipeManager_ErrorList.NoError;
		bError := FALSE;
	END_IF
END_IF

IF nErrorCode <> nRecipeManager_ErrorList.NoError AND nErrorCodeMemory <> nErrorCode THEN
	bError := TRUE;
END_IF
nErrorCodeMemory := nErrorCode;

// Update file name
IF iTableSelIndex <> iTableSelIndexMemory AND iTableSelIndex > 0 AND iTableSelIndex <= iMaxRecipeNumber THEN
	sRecipeName := astRecipeList[iTableSelIndex].sFileName;
	iTableSelIndexMemory := iTableSelIndex;
END_IF

IF bCopyPLC_2_TMP AND NOT bWritingRecipe AND NOT bReadingRecipe AND NOT bRefreshingRecipeList THEN
	MEMCPY(srcAddr := pPLC_Struct, destAddr := pTMP_PLC_Struct, n := UINT_TO_UDINT(uiPLC_StructSize));
	bCopyPLC_2_TMP := FALSE;
END_IF

IF (bCopyTMP_2_PLC AND bCopyTMP_2_PLC_Confirmed) AND NOT bWritingRecipe AND NOT bReadingRecipe AND NOT bRefreshingRecipeList THEN
	MEMCPY(srcAddr := pTMP_PLC_Struct, destAddr := pPLC_Struct, n := UINT_TO_UDINT(uiPLC_StructSize));
	bCopyTMP_2_PLC := bCopyTMP_2_PLC_Confirmed := FALSE;
END_IF
fbTON_Copy2PLCConfirmWindowReset(IN:= bCopyTMP_2_PLC, PT:= T#15S);
bCopyTMP_2_PLC R= fbTON_Copy2PLCConfirmWindowReset.Q;

ACTION ACT_DeleteRecipe:
CASE iStep OF
	0:	// Default Step
		bDeletingRecipe := TRUE;
		fbFileDelete(bExecute := FALSE);
		fbTON_StepTimeout(IN:= FALSE);
		iStep := 10;
		
	10: 	// Open file for read
		fbFileDelete(
			sPathName:= CONCAT(STR1:= sRecipesDirectory, STR2 := CONCAT(STR1:= sRecipeName ,STR2:= '.recipe')), 
			ePath:= PATH_GENERIC, 
			bExecute:= TRUE, 
			tTimeout:= T#1S, 
			bBusy=> , 
			bError=> , 
			nErrId=> );
		
		IF NOT fbFileDelete.bBusy THEN
			IF fbFileDelete.bError THEN
				iStep:= 99;
				uiErrorID:= fbFileDelete.nErrId;
				nErrorCode := nRecipeManager_ErrorList.FileDeleteError;
			ELSE
				iStep:= 50;
			END_IF
			fbFileDelete(bExecute:= FALSE); 
		END_IF
		
	50:		// Save success
		bRecipeDeleted_OK:= TRUE;
		iStep:= 100;
		
	99:
		bRecipeDeleted_OK:= FALSE;
		iStep:= 100;
		
	100:
		bDeletingRecipe := FALSE;
		fbTON_StepTimeout(IN:= FALSE);
		iStep:= 0;
END_CASE

fbTON_StepTimeout(IN:= TRUE, PT:= T#3S);
IF fbTON_StepTimeout.Q THEN
	fbTON_StepTimeout(IN:= FALSE);
	nErrorCode := nRecipeManager_ErrorList.DeleteRecipeTimeout;
	iStep:= 0;
	bDeletingRecipe := FALSE;
END_IF
END_ACTION

ACTION ACT_ReadRecipe:
CASE iStep OF
	0:	// Default Step
		bRecipeRead_OK:= FALSE;
		bReadingRecipe := TRUE;
		bCloseFileAfterError := FALSE;
		fbFileOpen(bExecute := FALSE);
		fbFileRead(bExecute := FALSE);
		fbFileClose(bExecute := FALSE);
		fbTON_StepTimeout(IN:= FALSE);
		bSizeNotEqual := FALSE;
		iStep := 10;
		
	10: 	// Open file for read
		fbFileOpen(
			sPathName:= CONCAT(STR1:= sRecipesDirectory, STR2 := CONCAT(STR1:= sRecipeName ,STR2:= '.recipe')), 
			nMode:= FOPEN_MODEREAD OR SEL(bTextFormat,FOPEN_MODEBINARY,FOPEN_MODETEXT), 
			ePath:= PATH_GENERIC, 
			bExecute:= TRUE, 
			tTimeout:= T#1S, 
			hFile=>hFiileHandler );
		
		IF NOT fbFileOpen.bBusy THEN
			IF fbFileOpen.bError THEN
				iStep:= 99;
				bFileOpen:=FALSE;
				uiErrorID:= fbFileOpen.nErrId;
				nErrorCode := nRecipeManager_ErrorList.FileOpenError;
			ELSE
				iStep:= 20;
				bFileOpen:=TRUE;
			END_IF
			fbFileOpen(bExecute:= FALSE); 
		END_IF
	
	20:		// Read Header
		fbFileRead(
			hFile:= hFiileHandler, 
			pReadBuff:= ADR(uiStructSize), 
			cbReadLen:= SIZEOF(uiStructSize), 
			bExecute:= TRUE, 
			tTimeout:= T#1S);
			
		IF NOT fbFileRead.bBusy THEN
			IF fbFileRead.cbRead <> fbFileRead.cbReadLen THEN
				nErrorCode := nRecipeManager_ErrorList.ReadSizeError;
				iStep:= 99;
			ELSE
				IF fbFileRead.bError THEN
					iStep:= 99;
					uiErrorID:= fbFileRead.nErrId;
					nErrorCode := nRecipeManager_ErrorList.ReadRecipeError;
				ELSE
					MEMSET(destAddr := pTMP_PLC_Struct, n := UINT_TO_UDINT(uiPLC_StructSize), fillByte := 0);		// clear memory before write data (necessary for CRC sum consistent)
					iStep:= 30;
				END_IF
			END_IF		
			fbFileRead(bExecute:= FALSE); 
		END_IF
		
	30:		// Read Data
		IF uiStructSize = uiPLC_StructSize THEN		// exact size data in recipe and PLC or not enought data in recipe
			fbFileRead.cbReadLen:= uiStructSize;
			bSizeNotEqual := FALSE;
		ELSIF uiStructSize < uiPLC_StructSize THEN
			fbFileRead.cbReadLen:= uiStructSize;
			bSizeNotEqual := TRUE;
		ELSE 	// to much data in recipe	 
			fbFileRead.cbReadLen:= uiPLC_StructSize;
			bSizeNotEqual := TRUE;
		END_IF
		fbFileRead(
			hFile:= hFiileHandler, 
			pReadBuff:= pTMP_PLC_Struct, 
			bExecute:= TRUE, 
			tTimeout:= T#1S);	
		IF NOT fbFileRead.bBusy THEN
			IF fbFileRead.cbRead <> fbFileRead.cbReadLen THEN
				iStep:= 99;
			ELSE
				IF fbFileRead.bError THEN
					iStep:= 99;
					uiErrorID:= fbFileRead.nErrId;
				ELSE
					iStep:= 35;
					wCRCsum:= F_DATA_TO_CRC16_CCITT(pData:= fbFileRead.pReadBuff, cbData := fbFileRead.cbReadLen, crc := 16#0000);
				END_IF
			END_IF
			fbFileRead(bExecute:= FALSE);		
		END_IF	
	
	35:		// Read and check CRC16sum	
		IF NOT bSizeNotEqual THEN
			fbFileRead(
				hFile:= hFiileHandler, 
				pReadBuff:= ADR(wCRCsumReaded), 
				cbReadLen := SIZEOF(wCRCsumReaded),
				bExecute:= TRUE, 
				tTimeout:= T#1S);	
			IF NOT fbFileRead.bBusy THEN
				IF fbFileRead.cbRead <> fbFileRead.cbReadLen THEN
					iStep:= 99;
					nErrorCode:= nRecipeManager_ErrorList.ReadSizeError;
				ELSE
					IF fbFileRead.bError THEN
						iStep:= 99;
						uiErrorID:= fbFileRead.nErrId;
					ELSE
						IF wCRCsumReaded = wCRCsum THEN
							iStep:= 40;
						ELSE
							iStep:= 99;
							nErrorCode:= nRecipeManager_ErrorList.BadCRC;
						END_IF
					END_IF
				END_IF
				fbFileRead(bExecute:= FALSE);		
			END_IF	
		ELSE
			iStep:= 40;
		END_IF
	
	40:		// Close file
			fbFileClose(
			hFile:= hFiileHandler, 
			bExecute:= TRUE, 
			tTimeout:= T#1S);
		IF NOT fbFileClose.bBusy THEN
			IF fbFileClose.bError THEN
				iStep:= 99;
				uiErrorID:= fbFileClose.nErrId;
				nErrorCode := nRecipeManager_ErrorList.FileCloseError;
			ELSE
				bFileOpen := FALSE;
				iStep:= 50;
			END_IF
			IF bCloseFileAfterError THEN
				bFileOpen R= NOT fbFileClose.bError;
				iStep:= 100;
				bCloseFileAfterError := FALSE;
			END_IF
			fbFileClose(bExecute:= FALSE);
		END_IF
		
	50:		// Save success
		bRecipeRead_OK:= TRUE;
		iStep:= 100;
		
	99:
		bRecipeRead_OK:= FALSE;
		IF bFileOpen THEN
			bCloseFileAfterError := TRUE;
			fbFileClose(bExecute:= TRUE); 
			iStep := 40;
		ELSE
			bCloseFileAfterError := FALSE;
			iStep:= 100;
		END_IF
		
	100:
		bReadingRecipe := FALSE;
		fbTON_StepTimeout(IN:= FALSE);
		fbFileOpen(bExecute := FALSE);
		fbFileRead(bExecute := FALSE);
		fbFileClose(bExecute := FALSE);
		iStep:= 0;
END_CASE

fbTON_StepTimeout(IN:= TRUE, PT:= T#3S);
IF fbTON_StepTimeout.Q THEN
	fbTON_StepTimeout(IN:= FALSE);
	nErrorCode := nRecipeManager_ErrorList.ReadRecipeTimeout;
	iStep:= 0;
	bReadingRecipe := FALSE;
END_IF
END_ACTION

ACTION ACT_RefreshRecipeList:

CASE iStep OF
	0:	// Default Step
		bRecipeList_Reloaded:= FALSE;
		bRefreshingRecipeList := TRUE;
		fbReloadRecipes(bExecute := FALSE);
		iStep := 10;
		iNbOfFoundRecipes := 0;
		MEMSET(destAddr := ADR(astRecipeList),n := SIZEOF(astRecipeList),fillByte := 0);
		fbReloadRecipes(
			eCmd:= eEnumCmd_First,
			sPathName:= CONCAT(STR1:= sRecipesDirectory, STR2:= '*.recipe'), 
			bExecute:= FALSE, 
			tTimeout:= T#2S, 
			bBusy=> , 
			bError=> , 
			nErrID=> , 
			bEOE=> , 
			stFindFile=> );
		fbTON_StepTimeout(IN:= FALSE);

	10: 	
		IF bAbort THEN
			bAbort := FALSE;
			fbReloadRecipes.eCmd := eEnumCmd_Abort;
			iStep := 30;
		ELSE
			iStep := 20;
		END_IF
		fbReloadRecipes(bExecute := FALSE);
		fbReloadRecipes(bExecute := TRUE);

	20:
		fbReloadRecipes(bExecute := FALSE);
		IF NOT fbReloadRecipes.bBusy THEN
			IF NOT fbReloadRecipes.bError THEN
				IF NOT fbReloadRecipes.bEOE THEN	
					IF iNbOfFoundRecipes <= iMaxRecipeNumber THEN	// Save entry and read next
						fbReloadRecipes.eCmd:= eEnumCmd_Next;
						iNbOfFoundRecipes := iNbOfFoundRecipes + 1;
						astRecipeList[iNbOfFoundRecipes].sFileName :=  LEFT(STR :=fbReloadRecipes.stFindFile.sFileName,SIZE := LEN(fbReloadRecipes.stFindFile.sFileName)-7);
						astRecipeList[iNbOfFoundRecipes].dtCreationTime := FILETIME_TO_DT(fbReloadRecipes.stFindFile.creationTime);						
					ELSE	// List  full
						bAbort := TRUE;
					END_IF
					iStep := 10;
				ELSE	// No more entries
					iStep := 30;
				END_IF
			ELSE	// log error
				uiErrorID := fbReloadRecipes.nErrID;
				iStep := 99;
			END_IF
		END_IF
			
	30:	// Save success
		bRecipeList_Reloaded:= TRUE;
		bRefreshingRecipeList := FALSE;
		iStep:= 0;
		
	99:
		bRecipeList_Reloaded:= FALSE;
		bRefreshingRecipeList := FALSE;
		iStep:= 0;
		
END_CASE
fbTON_StepTimeout(IN:= TRUE, PT:= T#5S);
IF fbTON_StepTimeout.Q THEN
	iStep:= 99;
END_IF
END_ACTION

ACTION ACT_WriteRecipe:
CASE iStep OF
	0:	// Default Step
		bRecipeSave_OK:= FALSE;
		bWritingRecipe := TRUE;
		fbTON_StepTimeout(IN:= FALSE);
		fbFileOpen(bExecute := FALSE);
		fbFileWrite(bExecute := FALSE);
		fbFileClose(bExecute := FALSE);
		IF uiPLC_StructSize < uiMaxStructureSize THEN
			uiStructSize := uiPLC_StructSize;
			iStep := 10;
		ELSE
			iStep := 99;
			nErrorCode :=nRecipeManager_ErrorList.StructToBig;
		END_IF
		
	10: 	// Open file for write
		fbFileOpen(
			sPathName:= CONCAT(STR1:= sRecipesDirectory, STR2 := CONCAT(STR1:= sRecipeName,STR2:= '.recipe')), 
			nMode:= FOPEN_MODEWRITE OR SEL(bTextFormat,FOPEN_MODEBINARY,FOPEN_MODETEXT), 
			ePath:= PATH_GENERIC, 
			bExecute:= TRUE, 
			tTimeout:= T#1S, 
			hFile=>hFiileHandler );
		
		IF NOT fbFileOpen.bBusy THEN
			IF fbFileOpen.bError THEN
				iStep:= 99;
				uiErrorID:= fbFileOpen.nErrId;
				nErrorCode := nRecipeManager_ErrorList.FileOpenError;
			ELSE
				iStep:= 20;
			END_IF
			fbFileOpen(bExecute:= FALSE);
		END_IF
		
	20:		// Save Header
		fbFileWrite(
			hFile:= hFiileHandler, 
			pWriteBuff:= ADR(uiStructSize), 
			cbWriteLen:= SIZEOF(uiStructSize), 
			bExecute:= TRUE, 
			tTimeout:= T#1S);
			
		IF NOT fbFileWrite.bBusy THEN
			IF fbFileWrite.cbWriteLen <> fbFileWrite.cbWrite THEN
				nErrorCode := nRecipeManager_ErrorList.WriteSizeError;
				iStep:= 99;
			ELSE
				IF fbFileWrite.bError THEN
					iStep:= 99;
					uiErrorID:= fbFileWrite.nErrId;
					nErrorCode := nRecipeManager_ErrorList.WriteRecipeError;
				ELSE
					iStep:= 30;
				END_IF
			END_IF	
			fbFileWrite(bExecute:= FALSE); 	
		END_IF
		
	30:		// Save Data
		IF bSavePLCStruct THEN
			fbFileWrite(pWriteBuff:= pPLC_Struct);
		ELSE
			fbFileWrite(pWriteBuff:= pTMP_PLC_Struct);
		END_IF
		fbFileWrite(
			hFile:= hFiileHandler, 
			cbWriteLen:= uiPLC_StructSize, 
			bExecute:= TRUE, 
			tTimeout:= T#1S);
		
		IF NOT fbFileWrite.bBusy THEN
			IF fbFileWrite.cbWriteLen <> fbFileWrite.cbWrite THEN
				nErrorCode := nRecipeManager_ErrorList.WriteSizeError;
				iStep:= 99;
			ELSE
				IF fbFileWrite.bError THEN
					iStep:= 99;
					uiErrorID:= fbFileWrite.nErrId;
					nErrorCode := nRecipeManager_ErrorList.WriteRecipeError;
				ELSE
					iStep:= 35;
					wCRCsum:= F_DATA_TO_CRC16_CCITT(pData:= fbFileWrite.pWriteBuff, cbData := fbFileWrite.cbWriteLen, crc := 16#0000);
				END_IF
			END_IF		
			fbFileWrite(bExecute:= FALSE); 
		END_IF
		
	35:		// calculate and write CRC check sum
		fbFileWrite(
			hFile:= hFiileHandler, 
			pWriteBuff:= ADR(wCRCsum), 
			cbWriteLen:= SIZEOF(wCRCsum), 
			bExecute:= TRUE, 
			tTimeout:= T#1S);
			
		IF NOT fbFileWrite.bBusy THEN
			IF fbFileWrite.cbWriteLen <> fbFileWrite.cbWrite THEN
				nErrorCode := nRecipeManager_ErrorList.WriteSizeError;
				iStep:= 99;
			ELSE
				IF fbFileWrite.bError THEN
					iStep:= 99;
					uiErrorID:= fbFileWrite.nErrId;
					nErrorCode := nRecipeManager_ErrorList.WriteRecipeError;
				ELSE
					iStep:= 40;
				END_IF
			END_IF		
			fbFileWrite(bExecute:= FALSE); 
		END_IF
		
	40:		// Close file
		fbFileClose(
			hFile:= hFiileHandler, 
			bExecute:= TRUE, 
			tTimeout:= T#1S,);
		IF NOT fbFileClose.bBusy THEN
			IF fbFileClose.bError THEN
				iStep:= 99;
				uiErrorID:= fbFileClose.nErrId;
				nErrorCode := nRecipeManager_ErrorList.FileCloseError;
			ELSE
				iStep:= 50;
			END_IF
			IF bCloseFileAfterError THEN
				bFileOpen R= NOT fbFileClose.bError;
				iStep:= 100;
				bCloseFileAfterError := FALSE;
			END_IF
			fbFileClose(bExecute:= FALSE);
		END_IF
		
	
	50:		// Save success
		bRecipeSave_OK:= TRUE;
		iStep:= 100;
	
	99:
		bRecipeSave_OK:= FALSE;
		IF bFileOpen THEN
			bCloseFileAfterError := TRUE;
			fbFileClose(bExecute:= TRUE); 
			iStep := 40;
		ELSE
			bCloseFileAfterError := FALSE;
			iStep:= 100;
		END_IF
		
	100:
		bWritingRecipe := FALSE;
		fbTON_StepTimeout(IN:= FALSE);
		fbFileOpen(bExecute := FALSE);
		fbFileWrite(bExecute := FALSE);
		fbFileClose(bExecute := FALSE);
		iStep:= 0;
END_CASE

fbTON_StepTimeout(IN:= TRUE, PT:= T#3S);
IF fbTON_StepTimeout.Q THEN
	fbTON_StepTimeout(IN:= FALSE);
	nErrorCode := nRecipeManager_ErrorList.WriteRecipeTimeout;
	iStep:= 0;
	bReadingRecipe := FALSE;
END_IF
END_ACTION

END_FUNCTION_BLOCK

// Common/SerialCom/fbSerialLinkCommunication
FUNCTION_BLOCK fbSerialLinkCommunication
VAR_IN_OUT
	RxBufferEL			: ComBuffer;	(* Receive data buffer; used with all receive function blocks *)
	TxBufferEL			: ComBuffer;	(* Transmit data buffer; used with all receive function blocks *)
END_VAR
VAR_OUTPUT
	bEL60CtrlError	: BOOL;
	eEL60CtrlErrorID	: ComError_t;
END_VAR
VAR
	fbEL60Ctrl		: SerialLineControl;
		(* 	I/O variables for a EL600* terminal*)
	stIn_EL60 AT %I*	: EL6inData22B;	(* linked to the EL6002 in the TwinCAT System Manager *)
	stOut_EL60 AT %Q*	: EL6outData22B;(* linked to the EL6002 in the TwinCAT System Manager *)
END_VAR


fbEL60Ctrl(
	Mode:= SERIALLINEMODE_EL6_22B,
	pComIn:= ADR(stIn_EL60), 
	pComOut:= ADR(stOut_EL60), 
	SizeComIn:=UINT_TO_INT( SIZEOF(stIn_EL60) ), 
	Error=> , 
	ErrorID=> , 
	TxBuffer:= TxBufferEL, 
	RxBuffer:= RxBufferEL);
IF fbEL60Ctrl.Error THEN
	bEL60CtrlError := TRUE;
	eEL60CtrlErrorID := fbEL60Ctrl.ErrorID;
END_IF

END_FUNCTION_BLOCK

// Common/String Functions/fbAcFormatString
FUNCTION_BLOCK fbAcFormatString
VAR_INPUT
	sFormat:STRING(255);
	sArg1:T_MaxString:= '';
	sArg2:T_MaxString:= '';
	sArg3:T_MaxString:= '';
	sArg4:T_MaxString:= '';
	sArg5:T_MaxString:= '';
	sArg6:T_MaxString:= '';
	sArg7:T_MaxString:= '';
	sArg8:T_MaxString:= '';
	sArg9:T_MaxString:= '';
	sArg10:T_MaxString:= '';
END_VAR
VAR_OUTPUT
	bError:BOOL;
	sOut:STRING(255);
END_VAR
VAR
	fbFormat:FB_FormatString;
	
	nErrorID: UDINT;
END_VAR

fbFormat(
	sFormat:= sFormat, 
	arg1:= F_STRING(sArg1), 
	arg2:= F_STRING(sArg2), 
	arg3:= F_STRING(sArg3), 
	arg4:= F_STRING(sArg4), 
	arg5:= F_STRING(sArg5), 
	arg6:= F_STRING(sArg6), 
	arg7:= F_STRING(sArg7), 
	arg8:= F_STRING(sArg8), 
	arg9:= F_STRING(sArg9), 
	arg10:= F_STRING(sArg10), 
	bError=> bError, 
	nErrId=> nErrorID, 
	sOut=> sOut);

END_FUNCTION_BLOCK

// Common/String Functions/fbConcatStrings
FUNCTION_BLOCK fbConcatStrings
VAR_INPUT
	Str1:STRING:= '';
	Str2:STRING:= '';
	Str3:STRING:= '';
	Str4:STRING:= '';
	Str5:STRING:= '';
	Str6:STRING:= '';
	Str7:STRING:= '';
	Str8:STRING:= '';
	
END_VAR
VAR_OUTPUT
	sOut:STRING;
END_VAR

IF LEN(STR := Str1) > 0 THEN
	sOut := Str1;
END_IF

IF LEN(STR := Str2) > 0 THEN
	sOut :=CONCAT (STR1 := sOut, STR2 := Str2);
END_IF

IF LEN(STR := Str3) > 0 THEN
	sOut :=CONCAT (STR1 := sOut, STR2 := Str3);
END_IF

IF LEN(STR := Str4) > 0 THEN
	sOut :=CONCAT (STR1 := sOut, STR2 := Str4);
END_IF

IF LEN(STR := Str5) > 0 THEN
	sOut :=CONCAT (STR1 := sOut, STR2 := Str5);
END_IF

IF LEN(STR := Str6) > 0 THEN
	sOut :=CONCAT (STR1 := sOut, STR2 := Str6);
END_IF

IF LEN(STR := Str7) > 0 THEN
	sOut :=CONCAT (STR1 := sOut, STR2 := Str7);
END_IF

IF LEN(STR := Str8) > 0 THEN
	sOut :=CONCAT (STR1 := sOut, STR2 := Str8);
END_IF

END_FUNCTION_BLOCK

// Common/String Functions/fDataToHexStr
FUNCTION fDataToHexStr : UINT
VAR_INPUT
	pData:POINTER TO BYTE;
	uiDataSize:UINT;
	pStr:POINTER TO BYTE;		// Wskaźnik na docelowy string
	uiStrSize: UINT;			// Rozmiar docelowego stringa
END_VAR
VAR
	i:UINT;
	sChar: STRING(2);
END_VAR

IF pData <> 0 AND uiDataSize > 0 AND uiStrSize >= (2*uiDataSize+3) THEN
	MEMSET(destAddr := pStr, n := uiStrSize, fillByte := 0);
	sChar := '0x';
	MEMCPY(srcAddr:= ADR(sChar), destAddr := pStr, n:= 2);	
	pStr := pStr+2;
	FOR i:= 1 TO uiDataSize DO
		sChar:= BYTE_TO_HEXSTR(in:=pData^, iPrecision:=2,bLoCase := FALSE);
		MEMCPY(srcAddr:= ADR(sChar), destAddr := pStr, n:= 2);
		pStr := pStr + 2;
		pData:=pData + 1;
	END_FOR
	fDataToHexStr := i;
END_IF

END_FUNCTION

// Common/String Functions/fGetStringUntil
FUNCTION fGetStringUntil : STRING
(**************************************************************
	Funkcja zwraca fragment stringa od początku stringa/zadanej pozycji do wybranego znaku;
	Przydatna do parsowania tekstu (np. wczytywania parametrów ze stringu)
**************************************************************)
VAR_INPUT
	sInput:STRING;
	iStartPos:INT:=0;
	sEndChar:STRING(1);
	bGetFromBegining: BOOL:= 0;		// If TRUE function returns string from begining of string, not from start pos
END_VAR
VAR
	i: INT;
	sChar:STRING(1);
END_VAR
VAR_OUTPUT
	iEndIndex:INT;
END_VAR

fGetStringUntil:='';
IF iStartPos > 0 AND iStartPos <= LEN(sInput) AND FIND(STR1 := sInput, STR2 := sEndChar)>0 THEN
	IF bGetFromBegining THEN	// Fill begining of output string with data
		fGetStringUntil := LEFT(STR:= sInput, SIZE:= iStartPos-1 );
	END_IF
	iEndIndex:= iStartPos;
	sChar := MID(STR:= sInput, LEN := 1, POS := iEndIndex);
	WHILE sChar <> sEndChar AND iEndIndex <= LEN(sInput) DO
		fGetStringUntil := INSERT( STR1 :=fGetStringUntil, STR2 := sChar, POS := LEN(STR:=fGetStringUntil));
		iEndIndex := iEndIndex +1;
		sChar := MID(STR:= sInput, LEN := 1, POS := iEndIndex);
	END_WHILE	
ELSE
	iEndIndex:= -1;	
END_IF

END_FUNCTION

// Common/String Functions/fHexStrToData
FUNCTION fHexStrToData : INT
VAR_INPUT
	sStr: STRING(2000);			// String postaci 0xFFFFFFF
	pData:POINTER TO BYTE;		// Wskaźnik na dane
	uiDataSize:UINT;			// Rozmiar danych
END_VAR
VAR
	i:UINT;
	pStr:POINTER TO BYTE;
	sChar: STRING(2);
END_VAR

pStr := ADR(sStr);
IF pData <> 0 AND uiDataSize > 0 AND LEN2(pStr)>2 THEN
	MEMSET(destAddr := pData, n := uiDataSize, fillByte := 0);
	MEMCPY(srcAddr:= pStr, destAddr := ADR(sChar), n:= 2);
	IF sChar = '0x' THEN
		pStr := pStr +2;		
	END_IF
	FOR i:= 1 TO uiDataSize DO
		MEMCPY(srcAddr:= pStr, destAddr := ADR(sChar), n:= 2);
		HEXSTR_TO_DATA(sHex:= sChar, pData :=pData, cbData := 1);
		pStr := pStr + 2;
		pData:=pData + 1;
	END_FOR
END_IF

END_FUNCTION

// Common/String Functions/fRemChar
FUNCTION fRemChar : STRING
(**************************************************************
	Funkcja usuwa ze stringu wybrany znak (np. znak spackji);

**************************************************************)
VAR_INPUT
	sInput:STRING;
	sCharToDelete:STRING(1);
END_VAR
VAR_OUTPUT
	bCharsRemoved:BOOL := FALSE;
END_VAR
VAR
	i: INT;
	sChar:STRING(1);
END_VAR

fRemChar := '';
IF FIND(STR1:= sInput, STR2:= sCharToDelete) > 0 THEN	// Przetwórz wejście tylko jeżeli jest w nim dany znak, jeśli nie pomiń przetwarzanie.
	FOR i := 1 TO LEN(sInput) DO
		sChar := MID(STR:= sInput, LEN := 1, POS := i);
		IF sChar <> sCharToDelete THEN
			fRemChar := INSERT( STR1 :=fRemChar, STR2 := sChar, POS := LEN(STR:=fRemChar));
		END_IF
	END_FOR	
	bCharsRemoved := TRUE;
ELSE
	bCharsRemoved := FALSE;
	fRemChar := sInput;
END_IF

END_FUNCTION

// Common/TimeProg/fbDateAndTimeCalc
FUNCTION_BLOCK PUBLIC fbDateAndTimeCalc
VAR_INPUT
	stData: REFERENCE TO stAircomTimeStruct;		// Opcjonalna obsługa dodatkowej struktury czasu
END_VAR
VAR_OUTPUT
END_VAR
VAR
	fbLocalSystemTime: FB_LocalSystemTime;
	bFirstCycle:BOOL:=TRUE;
	bSecond_Old:WORD;
	uiLastShiftNumber: UINT;
	tMemoryTime: TIME;
	fbFormatStr:FB_FormatString;
	{attribute 'is_connected' := 'stData'}
    bIsstDataConnected: BOOL;
END_VAR

fbLocalSystemTime(bEnable:=TRUE,dwCycle:=1);		// funkcja aktualizujaca czas zgodnie z systemowym sterownika

mCalculate(stData:= GVL_Aircom.stAC_DT_Data);		// Obliczanie zmiennych dla domyślnej struktury

IF bIsstDataConnected AND __ISVALIDREF(stData) THEN					// Obliczanie dla struktury dodatkowej
	stData := GVL_Aircom.stAC_DT_Data;
ELSE
	stData REF= 0;	
END_IF

METHOD INTERNAL mCalculate : BOOL
VAR_INPUT
	stData: REFERENCE TO stAircomTimeStruct;
END_VAR

VAR
	wMilliseconds: WORD;
END_VAR
// Określenie czasu cyklu sterownika
stData.tActualTime := TIME();
IF tMemoryTime <> T#0S THEN
	stData.tCycleTime:=stData.tActualTime- tMemoryTime;
	tMemoryTime := stData.tActualTime;
ELSE
	tMemoryTime := stData.tActualTime;	
END_IF

// Pobranie czasu do sterownika
stData.bTimeValid:= fbLocalSystemTime.bValid;								// Znacznik ważności daty
stData.stTimeStruct := fbLocalSystemTime.systemTime;				
stData.dtActualDate :=  SYSTEMTIME_TO_DT(TIMESTR := stData.stTimeStruct);	//


IF fbLocalSystemTime.bValid THEN 
	// Sygnalizacja nowej sekundy, minuty, godziny ... zmienne są zsynchronizowane z taskiem w którym są wykonywane!!!
	stData.bNew_Second_IMP := stData.stTimeStruct.wSecond <> bSecond_Old;
	IF stData.bNew_Second_IMP THEN		// Nowa sekunda
		stData.diPLC_UpTimeSeconds := stData.diPLC_UpTimeSeconds + 1; 
		stData.sTimeString := SYSTEMTIME_TO_STRING(stData.stTimeStruct);
		IF bFirstCycle THEN
			stData.wWeekNb := F_GetWeekOfTheYear(in:= stData.dtActualDate);				// Obliczanie nowego numeru tygodnia	
		END_IF
		IF stData.stTimeStruct.wSecond = 0 THEN		// Nowa minuta
			stData.bNew_Minute_IMP := TRUE;
			IF stData.stTimeStruct.wMinute = 0 THEN		// Nowa godzina
 				stData.bNew_Hour_IMP := TRUE;
				IF stData.stTimeStruct.wHour = 0 THEN		// Nowy dzień
					stData.bNew_Day_IMP := TRUE;
					IF stData.stTimeStruct.wDayOfWeek = 1 THEN		// Nowy tydzień
						stData.bNew_Week_IMP := TRUE;
						stData.wWeekNb := F_GetWeekOfTheYear(in:= stData.dtActualDate);				// Obliczanie nowego numeru tygodnia	
					END_IF
					IF stData.stTimeStruct.wDay = 1 THEN			// Nowy miesiąc
						stData.bNew_Month_IMP := TRUE;
						IF stData.stTimeStruct.wMonth = 1 THEN		// Nowy rok
							stData.bNew_Year_IMP := TRUE;
						END_IF
					END_IF
				END_IF
			END_IF
		END_IF
	ELSE
		stData.bNew_Second_IMP := stData.bNew_Minute_IMP := stData.bNew_Hour_IMP := stData.bNew_Day_IMP := stData.bNew_Week_IMP := stData.bNew_Month_IMP := stData.bNew_Year_IMP := FALSE;
	END_IF
	bSecond_Old := stData.stTimeStruct.wSecond;
	
	// Obsługa zmian
	stData.bNew_Shift := FALSE;
	IF stData.bNew_Hour_IMP OR bFirstCycle OR stData.uiShiftNumber < 1 OR stData.uiShiftNumber > 4 THEN
		IF stData.stTimeStruct.wHour >= 6 AND stData.stTimeStruct.wHour < 14 THEN
			stData.uiShiftNumber := 1;
		ELSIF stData.stTimeStruct.wHour >= 14 AND stData.stTimeStruct.wHour < 22 THEN
			stData.uiShiftNumber := 2;
		ELSIF stData.stTimeStruct.wHour >= 22 OR stData.stTimeStruct.wHour < 6 THEN
			stData.uiShiftNumber := 3;
		ELSE	
			stData.uiShiftNumber := 4;
		END_IF 
		stData.bNew_Shift := uiLastShiftNumber <> stData.uiShiftNumber AND NOT bFirstCycle;
		uiLastShiftNumber := stData.uiShiftNumber;
	END_IF
	IF bFirstCycle THEN
		stData.dtPLC_UpTime :=  stData.dtActualDate;
		bFirstCycle := FALSE;
	END_IF	
	//String for data logging
	wMilliseconds := stData.stTimeStruct.wMilliseconds/10;
	fbFormatStr(sFormat := '%0.2d-%0.2d %0.2d:%0.2d:%0.2d.%0.2d',
			arg1 := F_WORD(stData.stTimeStruct.wMonth), 
			arg2 := F_WORD(stData.stTimeStruct.wDay), 
			arg3 := F_WORD(stData.stTimeStruct.wHour),
			arg4 := F_WORD(stData.stTimeStruct.wMinute),
			arg5 := F_WORD(stData.stTimeStruct.wSecond),
			arg6 := F_WORD(wMilliseconds), sOut => stData.sLogTimeString);  
ELSE
	bSecond_Old := 0;
	stData.bNew_Second_IMP := stData.bNew_Minute_IMP := stData.bNew_Hour_IMP := stData.bNew_Day_IMP := stData.bNew_Week_IMP := stData.bNew_Month_IMP := stData.bNew_Year_IMP := FALSE;
END_IF
END_METHOD

END_FUNCTION_BLOCK

// Common/TimeTableStats/OOP_Version/fbTimeTable255
FUNCTION_BLOCK PUBLIC fbTimeTable255 IMPLEMENTS I_TimeTable255
VAR_INPUT
	rRowTime	: REAL;		// Time of actual table row
END_VAR
VAR
	astTT: ARRAY [1..50] OF stTimeStatsRow255;
	uiTTLastIndex:UINT:=1;
END_VAR

METHOD mPushRow		// Add Text and time to last timetable row
VAR_INPUT
	sText:STRING(255);
	rTimeValue:REAL;
END_VAR
MEMMOVE (srcAddr := ADR(astTT[1]), destAddr := ADR(astTT[2]), n := 49*SIZEOF(astTT[1]) );
astTT[1].rStepTime := rTimeValue;
astTT[1].sStepName := sText;
IF uiTTLastIndex < 50 THEN
	uiTTLastIndex := uiTTLastIndex + 1;	
END_IF
END_METHOD

METHOD mPushText		// Add Text to timetable row (time is added automatically from FB input)
VAR_INPUT
	sText:STRING(255);		// Text to save in timetable
END_VAR
MEMMOVE (srcAddr := ADR(astTT[1]), destAddr := ADR(astTT[2]), n := 49*SIZEOF(astTT[1]) );
astTT[1].rStepTime := rRowTime;
astTT[1].sStepName := sText;
IF uiTTLastIndex < 50 THEN
	uiTTLastIndex := uiTTLastIndex + 1;	
END_IF
END_METHOD

METHOD mReset
uiTTLastIndex := 0;
MEMSET(destAddr := ADR(astTT), fillByte := 0, n := 50*SIZEOF(astTT[1]));
END_METHOD

PROPERTY IsEmpty : BOOL	// Is Timetable empty?
GET
IsEmpty := uiTTLastIndex <= 0;
END_GET
END_PROPERTY

PROPERTY IsFull : BOOL		// Is Timetable full?
GET
IsFull := uiTTLastIndex >= 50;
END_GET
END_PROPERTY

PROPERTY LastIndex : UINT		// Last row in Timetable index?
GET
LastIndex := uiTTLastIndex;
END_GET
END_PROPERTY

END_FUNCTION_BLOCK

// Common/TimeTableStats/OOP_Version/I_TimeTable255
INTERFACE I_TimeTable255

METHOD mPushRow		// Add Text and time to last timetable row
VAR_INPUT
	sText:STRING(255);
	rTimeValue:REAL;
END_VAR
END_METHOD

METHOD mPushText		// Add Text to timetable row (time is added automatically from FB input)
VAR_INPUT
	sText:STRING(255);		// Text to save in timetable
END_VAR
END_METHOD

METHOD mReset	// Reset timetable
END_METHOD

PROPERTY IsEmpty : BOOL	// Is Timetable empty?
GET
END_GET
END_PROPERTY

PROPERTY IsFull : BOOL		// Is Timetable full?
GET
END_GET
END_PROPERTY

PROPERTY LastIndex : UINT		// Last row in Timetable index?
GET
END_GET
END_PROPERTY

END_INTERFACE

// Common/TimeTableStats/fbTimeTable
FUNCTION_BLOCK PUBLIC fbTimeTable IMPLEMENTS I_TimeTable
VAR CONSTANT
	uiMaxRows:UINT := 20;
END_VAR
VAR_INPUT
	rRowTime	: REAL;		// Time of actual table row
END_VAR
VAR
	astTimeTable: ARRAY [1..20] OF stTimeStatsRow;
	uiTTLastIndex:UINT:=1;	
END_VAR

METHOD mPushRow : BOOL
VAR_INPUT
	sText:STRING;
	rTimeValue:REAL;
END_VAR
MEMMOVE (srcAddr := ADR(astTimeTable[1]), destAddr := ADR(astTimeTable[2]), n := ((uiMaxRows-1)*SIZEOF(astTimeTable[1])) );
astTimeTable[1].rStepTime := rTimeValue;
astTimeTable[1].sStepName := sText;
IF uiTTLastIndex < uiMaxRows THEN
	uiTTLastIndex := uiTTLastIndex + 1;	
END_IF
END_METHOD

METHOD mPushText : BOOL		// Add Text to timetable row (time is added automatically from FB input)
VAR_INPUT
	sText:STRING;		// Text to save in timetable
END_VAR
MEMMOVE (srcAddr := ADR(astTimeTable[1]), destAddr := ADR(astTimeTable[2]), n := ((uiMaxRows-1)*SIZEOF(astTimeTable[1])) );
astTimeTable[1].rStepTime := rRowTime;
astTimeTable[1].sStepName := sText;
IF uiTTLastIndex < uiMaxRows THEN
	uiTTLastIndex := uiTTLastIndex + 1;	
END_IF
END_METHOD

METHOD mReset : BOOL
VAR_INPUT
END_VAR

VAR
END_VAR
uiTTLastIndex := 0;
MEMSET(destAddr := ADR(astTimeTable), fillByte := 0, n := SIZEOF(astTimeTable));
END_METHOD

PROPERTY IsEmpty : BOOL	// Is Timetable empty?
GET
IsEmpty := uiTTLastIndex <= 0;
END_GET
END_PROPERTY

PROPERTY IsFull : BOOL		// Is Timetable full?
GET
IsFull := uiTTLastIndex >= uiMaxRows;
END_GET
END_PROPERTY

PROPERTY LastIndex : UINT		// Last row in Timetable index?
GET
LastIndex := uiTTLastIndex;
END_GET
END_PROPERTY

PROPERTY MaxIndex : UINT		// Max row index in Timetable (max size)?
GET
MaxIndex := uiMaxRows;
END_GET
END_PROPERTY

END_FUNCTION_BLOCK

// Common/TimeTableStats/I_TimeTable
INTERFACE I_TimeTable

METHOD mPushRow : BOOL		// Add Text and time to last timetable row
VAR_INPUT
	sText:STRING;
	rTimeValue:REAL;
END_VAR
END_METHOD

METHOD mPushText : BOOL		// Add Text to timetable row (time is added automatically from FB input)
VAR_INPUT
	sText:STRING;		// Text to save in timetable
END_VAR
END_METHOD

METHOD mReset : BOOL	// Reset timetable
END_METHOD

PROPERTY IsEmpty : BOOL	// Is Timetable empty?
GET
END_GET
END_PROPERTY

PROPERTY IsFull : BOOL		// Is Timetable full?
GET
END_GET
END_PROPERTY

PROPERTY LastIndex : UINT		// Last row in Timetable index?
GET
END_GET
END_PROPERTY

PROPERTY MaxIndex : UINT		// Max row index in Timetable (max size)?
GET
END_GET
END_PROPERTY

END_INTERFACE

// Common/fbBlink
FUNCTION_BLOCK fbBlink
VAR_INPUT
	iBlinksQty:INT;
	tOn:TIME:=T#1S;
	tOff:TIME:=T#1S;
END_VAR
VAR_OUTPUT
	bQ:BOOL;
END_VAR
VAR
	fbTON_TactPulse:TON;
END_VAR

IF iBlinksQty > 0 THEN															
	fbTON_TactPulse(IN:= NOT fbTON_TactPulse.Q, PT:= SEL(bQ, tOff, tOn));		// Impuls at desired frequency (depends of bQ is TRUE or FALSE)
	bQ := bQ XOR fbTON_TactPulse.Q;												// Inverse output state
	IF NOT bQ AND fbTON_TactPulse.Q THEN										// Decrease Blinks nb after a full blink
 		iBlinksQty := iBlinksQty -1;
	END_IF	
END_IF

END_FUNCTION_BLOCK

// Common/fbLED_Blink
FUNCTION_BLOCK fbLED_Blink
VAR_IN_OUT	
	iBlinksQty:INT;
END_VAR
VAR_INPUT
	tOnTime:TIME:=T#1S;
	tOffTime:TIME:=T#1S;
END_VAR
VAR_OUTPUT
	bQ_LED:BOOL;
END_VAR
VAR
	fbTON_TactPulse:TON;
	bBlink: BOOL;
END_VAR

bBlink S= NOT bBlink AND iBlinksQty > 0 ;	// Rozpocznij cykl jeśli liczba mrugnięć większa od 0

IF bBlink THEN
	fbTON_TactPulse(IN:= NOT fbTON_TactPulse.Q, PT:= SEL(bQ_LED, tOffTime, tOnTime));		// Impuls co zadany czas
	bQ_LED := bQ_LED XOR fbTON_TactPulse.Q;		// Zmiana stanu wyjścia
	IF NOT bQ_LED AND fbTON_TactPulse.Q THEN	// Jeśli po mrugnięciu zmniejsz liczbę cykli i ew. zakończ mruganie
 		iBlinksQty := iBlinksQty -1;
		bBlink R= iBlinksQty = 0;
	END_IF	
END_IF

END_FUNCTION_BLOCK

// Common/fbOperationSynch
FUNCTION_BLOCK fbOperationSynch
VAR_INPUT
	bOperation1:BOOL;		// Impuls otwarcia lewej komory
	bOperation2:BOOL;		// Impuls otwarcia prawej komory
	tDelayTime:TIME;		// Czas różnicy
END_VAR
VAR_OUTPUT
	bZezwolenie:BOOL;
END_VAR
VAR
	bOperation1_MEM, bOperation2_MEM: BOOL;
	fbTON_ZezwoleniaL, fbTON_ZezwoleniaP: TON;
END_VAR

fbTON_ZezwoleniaL(IN:= NOT (bOperation1 AND NOT bOperation1_MEM), PT:= tDelayTime);
fbTON_ZezwoleniaP(IN:= NOT (bOperation2 AND NOT bOperation2_MEM), PT:= tDelayTime);
bOperation1_MEM := bOperation1;
bOperation2_MEM := bOperation2;
bZezwolenie := fbTON_ZezwoleniaL.Q AND fbTON_ZezwoleniaP.Q;

END_FUNCTION_BLOCK

// Common/fbPwmGenerator
FUNCTION_BLOCK PUBLIC fbPwmGenerator
VAR_INPUT
	bEnable:BOOL;	// Włącz generację impulsów
	rCycleInS:REAL;	// Okres impulsowania w sekundach
	rDutyCyclePercent:REAL;	// Wypełnienie impulsów 0..100%
END_VAR
VAR_OUTPUT
	bOutput:BOOL;	// Wyjście PWM
END_VAR
VAR
	fbTON:TON;
	rActualStateTime:REAL;
END_VAR

IF rDutyCyclePercent >= 100 THEN		// Jeśli zerowa moc wyłącz wyjście
	bOutput := bEnable;	
ELSIF rDutyCyclePercent <= 0 THEN		// Jeśli zerowa moc wyłącz wyjście
	bOutput := FALSE;
ELSE									// W sytuacjach pośrednich generuj odpowiedni cykl
	rActualStateTime:= rCycleInS*(SEL(bOutput,100-rDutyCyclePercent,rDutyCyclePercent)/100.0);
	fbTON(IN:= bEnable AND NOT fbTON.Q, PT:= REAL_TO_TIME(rActualStateTime*1000));
	bOutput := bEnable AND (bOutput XOR fbTON.Q);	
END_IF

END_FUNCTION_BLOCK

// Common/fbSequenceWork
FUNCTION_BLOCK fbSequenceWork
VAR_INPUT
	bEnable:BOOL;
	I_PimM1: I_PIM;			// Interfejs do I maszyny
	I_PimM2: I_PIM;			// Interfejs do II maszyny
END_VAR
VAR_OUTPUT
	bPermition_M1:BOOL;
	bPermition_M2:BOOL;	
END_VAR
VAR
	iWorkStep: INT;
	bM1_OperationEnded, bM1_OperationStatus, bM1_Test: BOOL;
	bM2_OperationEnded, bM2_OperationStatus, bM2_Test: BOOL;
	sM2_Rework:STRING(3);
END_VAR

I_PimM1.mGetStationData(bOperEnded => bM1_OperationEnded, bOperStatus => bM1_OperationStatus, bTestMode => bM1_Test );
I_PimM2.mGetStationData(bOperEnded => bM2_OperationEnded, bOperStatus => bM2_OperationStatus, bTestMode => bM2_Test, sOperRework =>sM2_Rework);

IF bEnable AND NOT bM1_Test AND NOT bM2_Test THEN
	CASE iWorkStep OF
	0:	// OKrok inicjalizacyjny
		bPermition_M1 := TRUE;
		bPermition_M2 := FALSE;
		iWorkStep := 1;
		
	1:	// Oczekiwanie na status OK z I maszyny
		IF bM1_OperationEnded AND bM1_OperationStatus THEN
			bPermition_M1 := FALSE;
			bPermition_M2 := TRUE;
			iWorkStep := 2;
		END_IF
		
	2:	// Oczekiwanie na status OK z II maszyny lub sygnał rework:false
		IF (bM2_OperationEnded AND bM2_OperationStatus) OR sM2_Rework = 'no' THEN
			bPermition_M1 := TRUE;
			bPermition_M2 := FALSE;
			iWorkStep := 1;	
		END_IF	
	ELSE 
		iWorkStep := 0;
	END_CASE
ELSE
	bPermition_M1 := bPermition_M2 := TRUE;
	iWorkStep := 0;
END_IF

END_FUNCTION_BLOCK

// PIM/Interfaces/I_PIM
INTERFACE I_PIM		// Interfejs implementowany przez blok PIMu - pozwala na pobranie odpowiednich danych z PIMu przez blok maszyny na stanowisku

// Zapis do DB danych rozszerzonych operacji - jeśli rozkaz dodany do kolejki zwraca TRUE, jeśli nie FALSE
METHOD m_SqlInsertExtendedData : BOOL		
VAR_INPUT
	pParameters: POINTER TO BYTE;				// Wskaźnik na tablicę elementów typu PIM_ExtDataRow
	uiArraySize: UINT;							// Rozmiar tablicy parametrów (może być pojedyncza zmienna)
END_VAR
END_METHOD

// Pobranie z DB statusu ostatniej operacji dla danego DM z poprzedniego stanowiska - gdy rozkaz zostanie wykonany zwraca TRUE
METHOD m_SqlSelLastOperationStatus : BOOL
VAR_INPUT
	sCodeDM:STRING(255);		// Identyfikator części (kod DataMatrix)
END_VAR
VAR_OUTPUT
	bProcessing:BOOL;			// Przetwarzanie rozkazu trwa (rozkaz dodany do kolejki)
	bResultOK:BOOL;				// Wynik wykonania rozkazu (do sprawdzenia gdy metoda zwróci TRUE)
	bPrevOperStat:BOOL;			// Status ostatniej operacji na poprzednim stanowisku
END_VAR
END_METHOD

 // Metoda zwraca strukturę do zapytania SQL uzupełnioną o dane z bloczka stanowiska
METHOD mGetStationData : stPIM_StationStatus
VAR_OUTPUT
	sCMD				: STRING;		// Zdarzenie jednostkowe/ rozkaz z PIMu np uaktualniono dane itp.
	bUserLogged			: BOOL;			// Użytkownik zalogowany
	bPIM_Active			: BOOL;			// Info o aktywności systemu PIM
	bTestMode			: BOOL;			// Aktywny tryb testowy
	bWorkPermittion		: BOOL;			// Informacja o zezwoleniu na pracę sumarycznie
	bWorkBlockPIM		: BOOL;			// Informacja o zezwoleniu na pracę z PIM
	bWorkBlockPLC		: BOOL;			// Informacja o zezwoleniu na pracę z PLC
	bConfirmation		: BOOL;			// Informacja o potwierdzeniu błędu
	bExternalMessage	: BOOL;			// Informacja o aktywnym komunikacie zewnętrznym
	nExtErrorClass		: nPIM_EventClasses;			// Informacja o aktywnym błędzie zewnętrznym
	bEventWaitInQueue	: BOOL;			// Info, że zdarzenie zewnętrzne czeka w kolejce
	nMachState			: nPIM_MachineStates;	// Aktualny status maszyny
	bOperInProgress		: BOOL;			// TRUE gdy operacja trwa
	bOperEnded			: BOOL;			// Impuls gdy operacja zakończona
	bOperStatus			: BOOL;			// Status ostatniej operacji
	nReworkSelected 	: nPIM_ReworkSelect;	// Operator wybrał Opcje reworku na tak lub nie
	nReoprtedNok 		: nPIM_ReportedNokSource;	// Operator zgłosił NOKa
END_VAR
END_METHOD

METHOD PUBLIC mNewEvent : BOOL
VAR_INPUT
	iEventId:	INT;				// Kod błędu w postaci inta (do przekonwertowania)
	nEventType: nPIM_EventClasses;	// ROdzaj nowego zdarzenia
	tMessageTime: TIME:= T#3S;		// Czas na wyświetlenie wiadomości- ma znaczenie tylko dla wiadomości (po tym czasie lub po starcie nowej operacji wiadomość znika)
END_VAR
END_METHOD

METHOD mNewServiceMessage : BOOL
VAR_INPUT
	sMessage: STRING(255);			// Wiadomośćdo wyświetlenia
	tMessageTime: TIME:= T#3S;		// Czas na wyświetlenie wiadomości- ma znaczenie tylko dla wiadomości (po tym czasie lub po starcie nowej operacji wiadomość znika)	
END_VAR
END_METHOD

// Masyzna zgłasza chęć przejścia do nowego stanu/kroku - pim wydaje zezwolenie na zmianę stanu dla poszczególnych kroków bazując na stanie z systemu PIM
METHOD mSetNewMachineState : BOOL
VAR_INPUT
	nMachineNewState: nPIM_MachineStates;		// Nowy stan maszyny
END_VAR
END_METHOD

PROPERTY PartsCtr_NOK : INT
GET
END_GET
END_PROPERTY

PROPERTY PartsCtr_OK : INT
GET
END_GET
END_PROPERTY

// The number of actually displayed error code ex "601"
PROPERTY prActiveErrorCode : STRING
GET
END_GET
END_PROPERTY

// Get CMD Value from PIM
PROPERTY prCMD : STRING
GET
END_GET
END_PROPERTY

// Get info 
PROPERTY prCurrentMachineState : nPIM_MachineStates
GET
END_GET
END_PROPERTY

// Get info 
PROPERTY prErrorClassExt : nPIM_EventClasses
GET
END_GET
END_PROPERTY

// Get info 
PROPERTY prErrorConfirmActive : BOOL
GET
END_GET
END_PROPERTY

// Get info 
PROPERTY prExternalEvtWaitInQueue : BOOL
GET
END_GET
END_PROPERTY

// Get info is PIM is active
PROPERTY prLastSavedStatus : BOOL
GET
END_GET
END_PROPERTY

// Get info is PIM is active
PROPERTY prNokReportedSource : nPIM_ReportedNokSource
GET
END_GET
END_PROPERTY

// Get info is PIM is active
PROPERTY prOperEnded : BOOL
GET
END_GET
END_PROPERTY

// Get info is PIM is active
PROPERTY prOperInProgress : BOOL
GET
END_GET
END_PROPERTY

// Get info is PIM is active
PROPERTY prPimActive : BOOL
GET
END_GET
END_PROPERTY

// Get info 
PROPERTY prPimBlockWork : BOOL
GET
END_GET
END_PROPERTY

// Get info 
PROPERTY prPlcBlockWork : BOOL
GET
END_GET
END_PROPERTY

// Get info is PIM is active
PROPERTY prReworkStatus : nPIM_ReworkSelect
GET
END_GET
END_PROPERTY

// Get info if station data is correctlly downloaded from database
PROPERTY prStationDataOK : BOOL
GET
END_GET
END_PROPERTY

// Get info is test mode is active
PROPERTY prTestMode : BOOL
GET
END_GET
END_PROPERTY

// Get info is user are logged?
PROPERTY prUserLogged : BOOL
GET
END_GET
END_PROPERTY

// Get info 
PROPERTY prWorkPermission : BOOL
GET
END_GET
END_PROPERTY

// Get info is that machine is EOL
PROPERTY prIsEol : BOOL
GET
END_GET
END_PROPERTY

// Get Station name followed by machine number ex: 'CA01PL19_1'
PROPERTY prPartCodeNumber : STRING(250)
GET
END_GET
END_PROPERTY

// Get Hidden status info
PROPERTY prIsHidden : BOOL
GET
END_GET
END_PROPERTY

// Get Line name ex: 'CA01PL'
PROPERTY prLineName : STRING(31)
GET
END_GET
END_PROPERTY

// Get Machine number
PROPERTY prMachNumber : INT
GET
END_GET
END_PROPERTY

// Get Station name followed by machine number ex: 'CA01PL19_1'
PROPERTY prStationAlias : STRING(31)
GET
END_GET
END_PROPERTY

// Get Station name ex: 'CA01PL19'
PROPERTY prStationName : STRING(31)
GET
END_GET
END_PROPERTY

END_INTERFACE

// Common/fbWriteStringToFile
FUNCTION_BLOCK fbWriteStringToFile
VAR_INPUT
	bWriteData:BOOL;
	sDataToWrite:STRING(255);
	sPath:STRING;
	sFilename:STRING;
END_VAR
VAR_OUTPUT
END_VAR
VAR
	iWriteStep: INT;
	fbOpenFile: FB_FileOpen;
	fbPutsFile:FB_FilePuts;
	fbCloseFile: FB_FileClose;
	hFileId: UINT;
END_VAR



CASE iWriteStep OF 
	0:	// Bezczynność - oczekiwanie na nowy zapis
		IF bWriteData THEN
			iWriteStep := 5;
		END_IF
		
	5:	// Sprawdzenie danych wejściowych
		IF sDataToWrite<> '' AND sPath <> '' AND sFilename <> '' THEN
			iWriteStep := 10;
			fbOpenFile(bExecute := FALSE);
 		END_IF
		
	10:	// Nowy zapis otwarcie pliku
		fbOpenFile(																								// Otwarcie pliku
			nMode:= FOPEN_MODEAPPEND OR FOPEN_MODETEXT, 
			ePath:= PATH_GENERIC, 
			sPathName := CONCAT (STR1 := sPath, STR2 := CONCAT(STR1:= sFilename, STR2:= '.csv')),
			bExecute:= TRUE, 
			tTimeout:= T#2S, 
			hFile=> hFileId);
		IF NOT fbOpenFile.bBusy THEN // AND fbOpenFile.bError THEN
			iWriteStep := 15;
			fbOpenFile(bExecute := FALSE);
			fbPutsFile(bExecute := FALSE);
		END_IF
		
	15:	// Zapisanie do pliku
		fbPutsFile(
			sNetId:= '',
			hFile:= hFileId,
			sLine:= sDataToWrite, 
			bExecute:= TRUE, 
			tTimeout:= T#1S);
		IF NOT fbPutsFile.bBusy THEN //AND fbPutsFile.bError THEN
			iWriteStep := 20;
			fbCloseFile(bExecute := FALSE);
			fbPutsFile(bExecute := FALSE);
		END_IF
		
	20:	// Zamykanie pliku
		fbCloseFile(																							// Zamknięcie pliku
			sNetId:= '', 
			hFile:= hFileId, 
			bExecute:= TRUE, 
			tTimeout:= T#2S);
		IF NOT fbCloseFile.bBusy THEN //AND fbCloseFile.bError THEN
			iWriteStep := 0;
			fbCloseFile(bExecute := FALSE);
		END_IF
	
	ELSE
	iWriteStep := 0;	
END_CASE

END_FUNCTION_BLOCK

// DataLoggers/fbTextDataLogger
FUNCTION_BLOCK fbTextDataLogger
VAR CONSTANT
	iMaxBufferSize:INT:= 30;
END_VAR
VAR_INPUT
	sNetId:T_MaxString;
	sDirectoryToSave:STRING;		// Katalog w którym zapisany będzie plik
	sFileNameWithFormat:STRING;		// Nazwa pliku do zapisu + rozszerzenie
	nMode:DWORD:= FOPEN_MODEAPPEND;		// Domyślnie FOPEN_MODEAPPEND, w bloczku dodane FOPEN_MODETEXT
	sPreambule:STRING;		// Znacznik dodawany na początku każdej linii (np. godzina, numer stanowiska itp)
	bSyncFile:BOOL;
	sCmdCommandToSync:BOOL;
END_VAR
VAR_OUTPUT
	bLoggerReady: BOOL;				// Gotowowy do zapisu danych
	bBufferEmpty: BOOL:= TRUE;		// Buffer wiadomości pusty
	bBufferFull: BOOL;				// Buffer wiadomości pełny
END_VAR
VAR
	asBufer:ARRAY[1..iMaxBufferSize] OF STRING[255];
	iBufferLastIndex:INT:= 0;
	
	iWorkStep: INT;
	fbFile_Open: FB_FileOpen;
	fbFile_Close: FB_FileClose;
	fbCreateDir: FB_CreateDir;
	fbPutsLine:	FB_FilePuts;
	fbNT_Ptocess: NT_StartProcess;
	bOpenTestPassed: BOOL;		// Zmienne do orzeczenia czy konfiguracja wejść jest OK
	
	sPath: STRING(255);
	hFileHandle: UINT;
	bSaveBuffor: BOOL;
	iSaveActLine: INT;
	sLineToSave: T_MaxString;
	bFileOpened: BOOL;
	bReInitFile: BOOL;
	sSyncCMD: STRING;
	fbTON_Reset: TON;
	sDirectoryToCreate: STRING;
	iStringCreateIndex: INT;
	sFileNameWithFormatMem:STRING;
END_VAR


IF bReInitFile OR sFileNameWithFormatMem <> sFileNameWithFormat THEN
	iWorkStep := 0;
	bReInitFile := FALSE;
	sFileNameWithFormatMem := sFileNameWithFormat;
END_IF

CASE iWorkStep OF
	0:	// Inicjalizacja po uruchomieniu
		fbTON_Reset(IN:= FALSE);
		bLoggerReady := FALSE;
		bBufferEmpty := TRUE;
		fbFile_Open(bExecute := FALSE);
		fbPutsLine(bExecute := FALSE);
		fbFile_Close(bExecute := FALSE);
		fbCreateDir(bExecute := FALSE);
		fbNT_Ptocess(START := FALSE);
		IF LEN(sDirectoryToSave) > 0 AND LEN(sFileNameWithFormat) > 0 THEN
			iWorkStep := 1;	
			iStringCreateIndex:= 1;
			IF RIGHT(STR := sDirectoryToSave, SIZE := 1) = '\' THEN
				sDirectoryToSave := LEFT(STR:= sDirectoryToSave, SIZE:= LEN(sDirectoryToSave)-1);
			END_IF
		END_IF
	
	1:	// Tworzenie drzewa katalogów
		sDirectoryToCreate := fGetStringUntil(sInput := sDirectoryToSave, iStartPos := iStringCreateIndex, sEndChar := '\', bGetFromBegining := TRUE, iEndIndex => iStringCreateIndex);
		IF iStringCreateIndex > 0 THEN
			iStringCreateIndex := iStringCreateIndex +1;	// Przesunięcie znacznika z bieżącego znalku
		END_IF 
		fbCreateDir(bExecute := FALSE);
		iWorkStep := 2;
	
	2: // Sprawdzenie czy są dane wejściowe
		IF sDirectoryToCreate <> '' THEN
			fbCreateDir( sNetId := sNetId,
				sPathName:= sDirectoryToCreate, 
				ePath:= E_OpenPath.PATH_GENERIC, 
				bExecute:= TRUE, 
				tTimeout:= T#2S);
			IF NOT fbCreateDir.bBusy THEN 
				IF ( NOT fbCreateDir.bError OR (fbCreateDir.bError AND (fbCreateDir.nErrId = 192 OR fbCreateDir.nErrId = 1827)) ) THEN	// Ścieżka istnieje lub została poprawnie utworzona
					iWorkStep := 1;
				ELSE
					iWorkStep := 90;
				END_IF
				fbCreateDir(bExecute := FALSE);
			END_IF	
		ELSE
			iWorkStep := 3;
		END_IF
 
	3: // Przygotowanie nazwy pliku
		IF RIGHT(STR:= sDirectoryToSave,SIZE := 1) <> '\' THEN
			sPath := CONCAT(STR1:= sDirectoryToSave, STR2:= CONCAT(STR1:= '\', STR2 := sFileNameWithFormat) ); 
		ELSE
			sPath := CONCAT(STR1:= sDirectoryToSave, STR2:= sFileNameWithFormat); 
		END_IF
		iWorkStep := 4;
		
	4:	// SPrawdzenie czy można otworzyć plik + konfiguracja bloczka wejściowego
		fbFile_Open( sNetId := sNetId,
			sPathName:= sPath, 
			nMode:= nMode OR FOPEN_MODETEXT, 
			ePath:= E_OpenPath.PATH_GENERIC, 
			bExecute:= TRUE, 
			tTimeout:= T#1S,
			hFile=> hFileHandle);
		IF NOT fbFile_Open.bBusy THEN
			IF NOT fbFile_Open.bError THEN
				bOpenTestPassed := TRUE;
				bFileOpened:= TRUE;
				iWorkStep := 5;
			ELSE
				iWorkStep := 90;
			END_IF
		END_IF
		
	5:	// Zamknięcie pliku po teście
		fbFile_Close( sNetId:= sNetId, 
			hFile:= hFileHandle, 
			bExecute:= TRUE, 
			tTimeout:= T#1S);
		IF NOT fbFile_Close.bBusy THEN
			IF fbFile_Close.bError THEN
				iWorkStep := 90;
			ELSE
				bFileOpened := FALSE;
				iWorkStep := 10;	
			END_IF
		END_IF
		
	10:	//	Gotowość na zapis
		bLoggerReady := TRUE;
		IF bSaveBuffor OR bBufferFull OR (iBufferLastIndex >= (iMaxBufferSize-5) AND mIsActEmpty()) THEN
			iSaveActLine := 1; 		
			fbFile_Open(bExecute := FALSE);
			fbPutsLine(bExecute := FALSE);
			fbFile_Close(bExecute := FALSE);
			iWorkStep := 15;
		END_IF
		
	15: // Sprawdzenie czy plik jest otwarty, ew. otwarcie pliku
		IF bFileOpened THEN
			iWorkStep := 20;
		ELSE 
			fbFile_Open(bExecute:= TRUE, 
				hFile=> hFileHandle);
			IF NOT fbFile_Open.bBusy THEN
				IF fbFile_Open.bError THEN
					iWorkStep := 90;
				ELSE
					bFileOpened := TRUE;
				END_IF
			END_IF
		END_IF
		
	20: // Zapis wszystkich linii
		IF iSaveActLine <= iBufferLastIndex AND iBufferLastIndex > 0 AND iSaveActLine <= iMaxBufferSize AND LEN(STR:= asBufer[iSaveActLine]) > 0 THEN
			sLineToSave := CONCAT(STR1:=asBufer[iSaveActLine], STR2:= '$n');
			fbPutsLine(bExecute := FALSE);
			iWorkStep := 25;
		ELSIF iSaveActLine >= iBufferLastIndex  THEN	// Zapis zakończony prawidłowo
			iBufferLastIndex := 0;
			bBufferEmpty := TRUE;
			bBufferFull := FALSE;
			MEMSET(destAddr:= ADR(asBufer), n := SIZEOF(asBufer), fillByte := 0);
			bSaveBuffor := FALSE;
			iWorkStep := 5;
		ELSIF iBufferLastIndex <0 OR iSaveActLine > iMaxBufferSize THEN		// Błędne parametry
			iWorkStep := 90;
		END_IF
		
	25:	// Zapis linii z bufora do pliku
		fbPutsLine( sNetId:= sNetId, 
			hFile:= hFileHandle, 
			sLine:= sLineToSave, 
			bExecute:= TRUE, 
			tTimeout:= T#200MS);
		IF NOT fbPutsLine.bBusy THEN
			IF fbPutsLine.bError THEN
				iWorkStep := 90;
			ELSE
				iSaveActLine := iSaveActLine + 1;
				iWorkStep := 20;
			END_IF
		END_IF
		
	30:	// Synchronizacja pliku z lokalizacją zewnętrzną
		sSyncCMD := 'xcopy ';
		sSyncCMD := CONCAT(STR1:= sSyncCMD, STR2:= sPath);
		sSyncCMD := CONCAT(STR1:= sSyncCMD, STR2:= '\');
		
		fbNT_Ptocess( NETID:= sNetId, 
			PATHSTR:= 'C:\Windows\System32', 
			DIRNAME:= 'C:\Windows\System32', 
			COMNDLINE:= 'xcopy c:\mysourcedirectory c:\mydestinationdirectory /I /E /Y /R', 
			START:= TRUE, 
			TMOUT:= , 
			BUSY=> , 
			ERR=> , 
			ERRID=> );
	
	90: // Błąd
		fbTON_Reset(IN:= TRUE, PT:= T#10S);
		IF fbTON_Reset.Q THEN
			fbTON_Reset(IN:= FALSE);
			iWorkStep := 0;
		END_IF
END_CASE

METHOD mAddLine : BOOL	// Metoda dodaje nową linię do zapisu lub zapełnia aktualną (jeśli aktualna jest pusta) i przechodzi dalej
VAR_INPUT
	sTextToSave:STRING;
END_VAR
IF LEN(sTextToSave) > 0 AND NOT bBufferFull THEN
	IF mIsActEmpty() THEN
		IF sPreambule <> '' THEN
			asBufer[iBufferLastIndex] := CONCAT(STR1:= sPreambule, STR2:= CONCAT(STR1:= '- ', STR2:= sTextToSave));	
		ELSE
			asBufer[iBufferLastIndex] := sTextToSave;
		END_IF
		iBufferLastIndex := LIMIT(1, iBufferLastIndex +1, iMaxBufferSize);
	ELSE
		iBufferLastIndex := LIMIT(1, iBufferLastIndex +1, iMaxBufferSize);
		IF sPreambule <> '' THEN
			asBufer[iBufferLastIndex] := CONCAT(STR1:= sPreambule, STR2:= CONCAT(STR1:= '- ', STR2:= sTextToSave));	
		ELSE
			asBufer[iBufferLastIndex] := sTextToSave;
		END_IF
	END_IF
	bBufferEmpty := FALSE;
	bBufferFull := iBufferLastIndex = iMaxBufferSize AND NOT mIsActEmpty();
	mAddLine := TRUE;	
ELSE 
	mAddLine := FALSE;
END_IF
END_METHOD

METHOD PUBLIC mAppendCurrentLine : BOOL
VAR_INPUT
	sAppendText:STRING;
	sAddSep:STRING(1):= '';			// Jeśli nie puste bloczek dodaje separator 
	bBreakLine:BOOL := FALSE;		// Jeśli true przesuwa znacznik na nową 'linię' (wiersz w buforze)
END_VAR
IF LEN(sAppendText) > 0 THEN
	
	IF mIsActEmpty() AND sPreambule <> '' THEN
		asBufer[iBufferLastIndex] := CONCAT(STR1:= sPreambule, STR2:= '- ');	
	END_IF
	asBufer[iBufferLastIndex] := CONCAT(STR1:= asBufer[iBufferLastIndex], STR2:= sAppendText);
	IF sAddSep <> '' THEN
		asBufer[iBufferLastIndex] := CONCAT(STR1:= asBufer[iBufferLastIndex], STR2:= sAddSep);
	END_IF
	bBufferEmpty := FALSE;
	IF bBreakLine AND NOT bBufferFull THEN
		iBufferLastIndex := LIMIT(1, iBufferLastIndex +1, iMaxBufferSize);
		bBufferFull := iBufferLastIndex = iMaxBufferSize AND NOT mIsActEmpty();
	END_IF
	mAppendCurrentLine := TRUE;	
END_IF
END_METHOD

METHOD mEndLine : BOOL
VAR_INPUT
END_VAR
IF iBufferLastIndex < iMaxBufferSize THEN
	iBufferLastIndex := LIMIT(1, iBufferLastIndex +1, iMaxBufferSize);
	bBufferFull := iBufferLastIndex = iMaxBufferSize AND NOT mIsActEmpty();
ELSE
	bBufferFull := mEndLine := TRUE;
END_IF
END_METHOD

METHOD PRIVATE mIsActEmpty : BOOL
VAR_INPUT
END_VAR
IF iBufferLastIndex < 1 THEN
	iBufferLastIndex := 1;
END_IF
mIsActEmpty := LEN(STR:= asBufer[iBufferLastIndex]) < 1;
END_METHOD

METHOD PUBLIC mSaveBuffor : BOOL
VAR_INPUT
END_VAR
mSaveBuffor:= bSaveBuffor:= TRUE;
END_METHOD

END_FUNCTION_BLOCK

// PIM/Interfaces/I_StationMachine
INTERFACE I_StationMachine	// Interfejs implementowany przez maszyny na stanowiskach - pozwala na kontrolę parametrów pracy maszyny

// Metoda TRUE kiedy dane wyjściowe są ok, jeśli nie FALSE (jeśli not bBusy i FALSE to błąd odczytu) 
METHOD mGetParamsData : BOOL
VAR_INPUT
	bTestParams:	BOOL;	// Jeśli TRUE metoda okresla czy ma dostęp do parametrów, jeśli tak zwraca TRUE, jeśli nie FALSE
END_VAR
VAR_OUTPUT
	bBusy:BOOL;		// Maszyna odświeża dane
	pMachineParametersStruct: POINTER TO BYTE;	// Wskaźnik do parametrów pracy maszyny
	uiMachineParametersSize: UINT;				// Rozmiar struktury parametrów pracy maszyny [bajty]
	wActualCRC16SumInMachine: WORD;				// Aktualna suma CRC16 obliczona z parametrów
END_VAR
END_METHOD

END_INTERFACE

// PIM/POUs/fbPIM_Dummy
FUNCTION_BLOCK fbPIM_Dummy IMPLEMENTS  I_PIM
VAR_IN_OUT
	stPimInOut:stPIM_ServiceInOuts;				// Dane pobierane z/ wysyłane do systemu PIM
END_VAR
VAR_INPUT
	bSaveStatus: BOOL;
	bStatusToSave: BOOL;
	iStatusErrCode: INT;
END_VAR
VAR_OUTPUT
	bUserLogged: BOOL;
	bWorkPermitt: BOOL;
END_VAR
VAR
	nExtEvent: nPIM_EventClasses;
	fbTON_Reset: TON;
	nMachineState: nPIM_MachineStates;
	fbTON_UserLogedDeleyed: TON;
	fbRTrig_StatusSave: R_TRIG;
END_VAR

fbTON_Reset(IN:= stPimInOut.bConfirmEvent, PT:= T#1S);
stPimInOut.bConfirmEvent R= fbTON_Reset.Q;

fbTON_UserLogedDeleyed(IN:= stPimInOut.bUSerLogged, PT:= T#200MS, Q=> bUserLogged);

bWorkPermitt := stPimInOut.bTestMode OR NOT stPimInOut.bPIMActive OR 
					(fbTON_UserLogedDeleyed.Q AND NOT stPimInOut.bWorkBlock_PIM AND NOT stPimInOut.bWorkBlock_PLC
					AND (NOT stPimInOut.bAlarmPLC OR stPimInOut.bNonBlockingAlarm) );

(* Zapis do DB danych rozszerzonych operacji - jeśli rozkaz dodany do kolejki zwraca TRUE, jeśli nie FALSE*)
METHOD m_SqlInsertExtendedData : BOOL
VAR_INPUT
	(* Struktura zapytania i danych do zapytania odpowiednio uzupełniona*)
//	stDataStruct	: stSQL_QueryParamsStruct;
	(* Zapytanie SQL do zapisu (do dostosowania liczba zapisanych danych)*)
	sSQLCmd	: STRING(1000);
END_VAR
m_SqlInsertExtendedData := TRUE;
END_METHOD

// Pobranie z DB statusu ostatniej operacji dla danego DM z poprzedniego stanowiska - gdy rozkaz zostanie wykonany zwraca TRUE
METHOD m_SqlSelLastOperationStatus : BOOL
VAR_INPUT
	sCodeDM:STRING(255);		// Identyfikator części (kod DataMatrix)
END_VAR
VAR_OUTPUT
	bProcessing:BOOL;			// Przetwarzanie rozkazu trwa (rozkaz dodany do kolejki)
	bResultOK:BOOL;				// Wynik wykonania rozkazu (do sprawdzenia gdy metoda zwróci TRUE)
	bPrevOperStat:BOOL;			// Status ostatniej operacji na poprzednim stanowisku
END_VAR
bProcessing:= FALSE;
bResultOK:= TRUE;
bPrevOperStat:=TRUE;
m_SqlSelLastOperationStatus := TRUE;
END_METHOD

// Metoda zwraca strukturę do zapytania SQL uzupełnioną o dane z bloczka stanowiska
METHOD mGetStationData : stPIM_StationStatus
VAR_OUTPUT
	sCMD			: STRING;		// Zdarzenie jednostkowe/ rozkaz z PIMu np uaktualniono dane itp.
	bUserLogged		: BOOL;			// Użytkownik zalogowany
	bPIM_Active		: BOOL;			// Info o aktywności systemu PIM
	bTestMode		: BOOL;			// Aktywny tryb testowy
	bWorkPermittion	: BOOL;			// Informacja o zezwoleniu na pracę z PIM
	bConfirmation	: BOOL;			// Informacja o potwierdzeniu błędu
	bExternalMessage: BOOL;			// Informacja o aktywnym komunikacie zewnętrznym
	nExtErrorClass	: nPIM_EventClasses;			// Informacja o aktywnym błędzie zewnętrznym
	nMachState		: nPIM_MachineStates;	// Aktualny status maszyny
	bOperInProgress	: BOOL;			// TRUE gdy operacja trwa
	bOperEnded		: BOOL;			// Impuls gdy operacja zakończona
	bOperStatus		: BOOL;			// Status ostatniej operacji
	sOperRework		: STRING(3);	// Status wyboru reworku na true zmienna przyjmuje wartości 'yes' lub 'no'. Jeśli pusta brak wyboru
END_VAR
sCMD:= stPimInOut.sCmdPIM2PLC;
bUserLogged:= stPimInOut.bUSerLogged;
bPIM_Active:= stPimInOut.bPIMActive;
bTestMode := stPimInOut.bTestMode;
bWorkPermittion := bWorkPermitt;
nExtErrorClass := nExtEvent;
bExternalMessage := FALSE;
nMachState := nMachineState;
bOperInProgress:= bOperEnded:=bOperStatus := FALSE;
sOperRework := '';
END_METHOD

METHOD PUBLIC mNewEvent : BOOL
VAR_INPUT
	iEventId:	INT;				// Kod błędu w postaci inta (do przekonwertowania)
	nEventType: nPIM_EventClasses;	// ROdzaj nowego zdarzenia
	tMessageTime: TIME:= T#3S;		// Czas na wyświetlenie wiadomości- ma znaczenie tylko dla wiadomości (po tym czasie lub po starcie nowej operacji wiadomość znika)
END_VAR
IF nEventType <> nPIM_EventClasses.Message THEN
	nExtEvent := nEventType;	
END_IF
END_METHOD

{warning 'add method implementation '}
METHOD mNewServiceMessage : BOOL
VAR_INPUT
	(* Wiadomośćdo wyświetlenia*)
	sMessage	: STRING(255);
	(* Czas na wyświetlenie wiadomości- ma znaczenie tylko dla wiadomości (po tym czasie lub po starcie nowej operacji wiadomość znika)	*)
	tMessageTime	: TIME := TIME#3s0ms;
END_VAR
nExtEvent := nPIM_EventClasses.Message;
END_METHOD

(* Masyzna zgłasza chęć przejścia do nowego stanu/kroku - pim wydaje zezwolenie na zmianę stanu dla poszczególnych kroków bazując na stanie z systemu PIM*)
METHOD mSetNewMachineState : BOOL
VAR_INPUT
	(* Nowy stan maszyny*)
	nMachineNewState	: nPIM_MachineStates;
END_VAR
IF nMachineNewState = nPIM_MachineStates._9_ResetInProgress THEN
	mSetNewMachineState := stPimInOut.bConfirmEvent;
ELSIF nMachineNewState = nPIM_MachineStates._0_Standby_NotReady THEN
	nExtEvent := nPIM_EventClasses.NoError;
	mSetNewMachineState := TRUE;
ELSE
	mSetNewMachineState := TRUE;
END_IF
IF mSetNewMachineState THEN
	nMachineState := nMachineNewState;	
END_IF
END_METHOD

END_FUNCTION_BLOCK

// PIM/POUs/fbPIM_MachineDummy
// Machine for PIM FB testing
FUNCTION_BLOCK fbPIM_MachineDummy IMPLEMENTS I_StationMachine
VAR_IN_OUT
END_VAR
VAR_INPUT
END_VAR
VAR_OUTPUT
	nError:nPIM_ErrorCodes;
END_VAR
VAR
	I_PimSystem			: I_PIM;		// PIM Interface
	iWorkStep: INT;
	bNewOper: BOOL;
	bNoWorkPermition: BOOL;
	bNewAlarm: BOOL;
	bNewError: BOOL;
	bServiceReset: BOOL;
	fbTON_Delay: TON;
END_VAR



CASE iWorkStep OF 
	0:	// Initial
		I_PimSystem.mSetNewMachineState(nMachineNewState := nPIM_MachineStates._0_Initialization);
		I_PimSystem.mSetNewMachineState(nMachineNewState := nPIM_MachineStates._0_Standby_NotReady);
		iWorkStep := 10;
		
	10: 
		I_PimSystem.mSetNewMachineState(nMachineNewState := nPIM_MachineStates._2_ReadyForNewOperation);
		IF bNewOper THEN
			bNoWorkPermition:= FALSE;
			IF I_PimSystem.mSetNewMachineState(nMachineNewState := nPIM_MachineStates._3_NewOperationStarted) THEN
				iWorkStep := 15;
			ELSE
				bNoWorkPermition:= TRUE;
			END_IF
		ELSIF bNewAlarm THEN
			bNewAlarm := FALSE;
		ELSIF bNewError THEN
			bNewError:= FALSE;	
		END_IF
		
	90:	// Błąd aktywny
		I_PimSystem.mSetNewMachineState(nMachineNewState := nPIM_MachineStates._8_WaitForReset);
		IF bServiceReset OR I_PimSystem.mSetNewMachineState(nMachineNewState := nPIM_MachineStates._9_ResetInProgress) THEN
			bServiceReset := FALSE;
			iWorkStep := 95;
		END_IF
		
	95:	// Reset
		fbTON_Delay(IN:= TRUE, PT:= T#1S);
		IF bNewError THEN
			mNewEvent(nEvent:=nPIM_ErrorCodes.UnKnownLock , nEventClass := nPIM_EventClasses.Error);
		ELSIF bNewAlarm THEN
			mNewEvent(nEvent:=nPIM_ErrorCodes.UnKnownAlarm , nEventClass := nPIM_EventClasses.Alarm);
		ELSE
			I_PimSystem.mSetNewMachineState(nMachineNewState := nPIM_MachineStates._0_Standby_NotReady);
			iWorkStep := 10;
		END_IF
		bNewAlarm := bNewError :=FALSE;
	
END_CASE

METHOD FB_init : BOOL
VAR_INPUT
	bInitRetains : BOOL; // if TRUE, the retain variables are initialized (warm start / cold start)
	bInCopyCode : BOOL;  // if TRUE, the instance afterwards gets moved into the copy code (online change)I_Pim
	I_Pim	: I_PIM;		// Interfejs do bloku PIM
END_VAR
I_PimSystem := I_Pim;
END_METHOD

(* Metoda TRUE kiedy dane wyjściowe są ok, jeśli nie FALSE (jeśli not bBusy i FALSE to błąd odczytu) *)
METHOD mGetParamsData : BOOL
VAR_INPUT
	bTestParams:	BOOL;	// Jeśli TRUE metoda okresla czy ma dostęp do parametrów, jeśli tak zwraca TRUE, jeśli nie FALSE
END_VAR
VAR_OUTPUT
	bBusy	: BOOL;										//	Maszyna odświeża dane
	pMachineParametersStruct	: POINTER TO BYTE;		// 	Wskaźnik do parametrów pracy maszyny
	uiMachineParametersSize	: UINT;						// 	Rozmiar struktury parametrów pracy maszyny [bajty]
	wActualCRC16SumInMachine	: WORD;					//	Aktualna suma CRC16 obliczona z parametrów
END_VAR
IF bTestParams THEN
	mGetParamsData := FALSE;
ELSE
	pMachineParametersStruct := 0;
	uiMachineParametersSize := 0;
	wActualCRC16SumInMachine := F_DATA_TO_CRC16_CCITT(pData := pMachineParametersStruct, cbData := uiMachineParametersSize, crc := 16#0000);
	bBusy := FALSE;
	mGetParamsData := TRUE;
END_IF
END_METHOD

METHOD INTERNAL mNewEvent : BOOL
VAR_INPUT
	nEventClass:nPIM_EventClasses;
	nEvent: nPIM_ErrorCodes;
END_VAR
IF nEventClass = nPIM_EventClasses.AlarmAutoConfirm OR nEventClass = nPIM_EventClasses.Message THEN		// Alarm nieblokadowy
	I_PimSystem.mSetNewMachineState(nPIM_MachineStates._0_Initialization);
	iWorkStep := 95;
ELSE
	I_PimSystem.mSetNewMachineState(nPIM_MachineStates._7_ErrorOccurr);
	I_PimSystem.mNewEvent(iEventId := nEvent, nEventType := nEventClass, tMessageTime := T#0S);
	iWorkStep := 90;
END_IF
nError := nEvent;
END_METHOD

END_FUNCTION_BLOCK

// PIM/POUs/fbPIM_SimplePimStation
FUNCTION_BLOCK FINAL fbPIM_SimplePimStation IMPLEMENTS  I_SqlCmds
VAR_INPUT
	stPimInOut: REFERENCE TO stPIM_ServiceInOuts;	// Dane pobierane z/ wysyłane do systemu PIM
	sLineName : STRING(31);							// Nazwa linii w systemie PIM
	sStationName : STRING(31);						// Nazwa stanowiska w systemie PIM
	iMachineNumber : INT:= 1;					// Numer maszyny na stanowisku
	bIsHidden : BOOL:= FALSE;					// Czy ukrywanie zapisu statusu (jeśli TRUE część nie jest liczona jako wyjściowa ze stanowiska)
	sPrevStationName : STRING(31);			// Do sprawdzenia statusu ostatniej operacji - jeśli funkcja nieużywana zostaw puste
	stStationSettings:stPIM_StationSettings;	// Ustawienia stanowiska	
	bSaveStatus: BOOL;							// Zbocze narastające powoduje wyzwolenie zapisu statusu
	bStatusToSave: BOOL;						// Status do zapisania
	iEventId:	INT;							// Kod błędu w postaci inta (do przekonwertowania)
	nEventType: nPIM_EventClasses;				// ROdzaj nowego zdarzenia
	sMessage: STRING(255);						// Wiadomośćdo wyświetlenia
	tMessageTime: TIME:= T#3S;					// Czas na wyświetlenie wiadomości- ma znaczenie tylko dla wiadomości (po tym czasie lub po starcie nowej operacji wiadomość znika)	
END_VAR
VAR_OUTPUT
	bStationDataOK: BOOL;
	bUserLogged: BOOL;							// Użytkownik zalogowany
	bTestMode: BOOL;
	bWorkPermitt: BOOL;
	bStationReady: BOOL;
	nErrorID:INT;
	bResetSignal: BOOL;
	stStationStatus: stPIM_StationStatus;
	nReoprtedNokSource: nPIM_ReportedNokSource;
	nReworkMenuStatus:nPIM_ReworkSelect;
END_VAR
VAR
	I_SqlCore:	I_SQL_Core;						// Interfejs do obsługi zapytań SQL
	bPIM_Working:BOOL;							// Informacja o działaniu systemu PIM (Odświeżany Cykliczny lifeBit)
	nActEventClass: nPIM_EventClasses;
	nMachineState: nPIM_MachineStates;
	iWorkStep :INT;
	stSqlComandData:stSQL_ClientNode;			// Struktura do zapytań z danymi powrotnymi (struktura jest blokowana na czas zapytania)
	stSqlComandDataTMP:stSQL_ClientNode;		// Struktura do zapytań bez danych powrotnych (podczas tworzenia zapytania dynamicznie tworzona kopia)
	bSelectStationId, bInsertStatus, bSelPreviousStatus, bSelMachineParamsData, bInsMachineParamsData, bSelMachineParamsCRC: BOOL;
	bReturnDataBusy: BOOL;
	liLPartStatusId: LINT;
	stRetDataLineStation	: stSQL_RetDataProdLineStat;	
	stRetDataMachParams		: stSQL_RetDataProdMachParams;	
	stRetDataUserRole		: stSQL_RetDataUserRole;
	iConvTMP:INT;
	bCmdAddError: BOOL;
	bCmdSended: BOOL;
	bPimCmdProcessing: BOOL:= FALSE;
	sActCmd: STRING;
	fbTOF_PimWorking: TOF;
	asUnsuportedCmds:ARRAY [1..5] OF STRING;
	bReturnDataReserved_StationId, bReturnDataReserved_InsOperStat, bReturnDataReserved_InsStatusExtData, bReturnDataReserved_SelLastOperStat,
		bReturnDataReserved_SelMachParams, bReturnDataReserved_InsMachParams, bReturnDataReserved_SelMachParamsCRC: BOOL;		// Zmienne rezerwujące strukturę danych dla zapytań które zwracają dane z DB
	diMachineParamsInsertId: DINT;
	bUpdateData: BOOL;
	fbRTRIG_UserLogged: R_TRIG;
	fbTON_ConfirmReset: TON;
	wCrcSumInDb:WORD;
	bMachineParamsOK: BOOL;
	bMachParSql_Processing: BOOL;
	bMachParSql_Result_OK: BOOL;
	diLastParamsInsID: DINT;
	sStringToParse: STRING(255);
	bCmdReaded:BOOL;
	
	sUserRole: STRING;
	sUserLang: STRING(3);
	fbTON_MessageTimer, fbTON_ServiceMessageTimer:TON;	// TImer wyświetlania alarmu lub wiadomości w dolnym pasku
		
	bLockAfterStatusSave: BOOL;
	
	bNewOperationInProgress: BOOL;		// Inforamcja o rozpoczętej operacji, kasowana po zakończeniu operacji i zapisie statusu operacji
	bStatusSaveTriggered: BOOL;		// Flaga o wystawieniu zapisu statusu do DB
	bStatusSavedOK: BOOL;				// Informacja o poprawnym zapisie statusu
	bOperationEndedError: BOOL;			// Informacja, że operacja zakończyła się błędem
	bPreviousOperationStatus: BOOL;
	
	wCrcSumInMachine: WORD;
	bSQLCmdError: BOOL;
	bStationDataOK_Temp: BOOL;
	iPartsQtyPermittTemporary: INT;
	bParReadBusy: BOOL;
	pParametersPtr: POINTER TO BYTE;
	uiParametersSize: UINT;
	bMachParamsSendToDB, bMachParamsReadFromDB: BOOL;	// Zapis/odczyt parametrów pracy maszyny do/z bazy danych

	
	bParamsInMachineUpdated: BOOL;
	bRetool: BOOL;
	iOutBoxQty,	iOutBoxTargetQty: INT;
	bRefreshData: BOOL;
	sCmdToSendToMachine: STRING;
	fbTON_AutoReset: TON;
	iMemPimWorkStep: INT;
	aiPimWorkStepHistoric: ARRAY [1..10] OF INT;
	fbLogger:fbTextDataLogger;
	sFormat:STRING(1023);
	fbFormatStr2:FB_FormatString2;
	fbFormatStr:FB_FormatString;

	iCtr_Operations, iCtr_OperationsInterrupted, iCtr_OperationsEndedOK, iCtr_OperEndedOK_Method, iCtr_OperationsEndedNOK: INT;
	iCtr_PIM_PartsOK, iCtr_PIM_PartsNOK, iCtr_PIM_ReworkYes, iCtr_PIM_PartOK_SaveError, iCtr_PIM_PartNOK_SaveError, iCtr_StatusSaveOK, iCtr_StatusSaveError, iCtr_Errors: INT;
	iCtrMem_Operations, iCtrMem_OperationsInterrupted, iCtrMem_OperationsEndedOK, iCtrMem_OperEndedOK_Method, iCtrMem_OperationsEndedNOK: INT;
	iCtrMem_PIM_PartsOK, iCtrMem_PIM_PartsNOK, iCtrMem_PIM_ReworkYes, iCtrMem_PIM_PartOK_SaveError, iCtrMem_PIM_PartNOK_SaveError, iCtrMem_StatusSaveOK, iCtrMem_StatusSaveError, iCtrMem_Errors: INT;
	bWriteHistoricData: BOOL;
	bTestZapisu: BOOL;
	bOperationEnded: BOOL;
	bOperationStatus: BOOL;
	fbTON_UserLogedDeleyed: TON;
	bStatusToSaveMemory: BOOL;
	bStationIdValid: BOOL;
	bLastStatus: BOOL;
	sLastErrCode: STRING(10);
	sLastDMCode: STRING(255);
	fbTON_CmdHangedUp: TON;
	uiCtr_CmdReset: UINT;
	fbTON_CmdPLC2PIM_Reset: TON;
	bCmdPlc2PimSended: BOOL;
	sCmdPlc2PimBufer: STRING(255);
END_VAR
VAR PERSISTENT
	liIdOutCompossedPartMemory:LINT;			// Id ostatniego elementu składanego na stanowisku z zatwierdzonymi parametrami
	wLastParametersCrcMemory: WORD;			// Suma CRC ostatnich zgodnych parametrów
END_VAR

(*	Funkcjonalności do zapewnienia: 
	-* Obsługa syganłu zezwolenia na pracę	
	-* Zliczanie części i obsługa Reworku
	-* Możliwość wyświetlenia alarmów oraz ich reset 
	-* Zapis statusu operacji
	- Zapis danych rozszerzonych
	- Zapis dodatkowych danych
	-* Kontrola parametrów maszyny
	- Automatyczne przezbrojenie
	
	Wymagania - możliwie uniwersalny interfejs między stacją <-> maszyną + reguła DRY
*)


fbRTRIG_UserLogged(CLK := stPimInOut.bUSerLogged);
fbTON_UserLogedDeleyed(IN:= stPimInOut.bUSerLogged, PT:= T#200MS, Q=> bUserLogged);
fbLogger(sNetId := '', sPreambule := GVL_Aircom.stAC_DT_Data.sTimeString);
bRefreshData S= fbRTRIG_UserLogged.Q;
bTestMode := stPimInOut.bTestMode;

IF NOT stPimInOut.bPIMActive AND NOT (iWorkStep <> -1) THEN
	iWorkStep := -1;
	stPimInOut.sPlcServiceMessage := 'PIM_NotActive';
	fbTON_ServiceMessageTimer.IN:= FALSE;
	fbTON_AutoReset(IN:= nMachineState = nPIM_MachineStates._8_WaitForReset , PT:= T#5S);
END_IF

IF iMemPimWorkStep <> iWorkStep THEN
	MEMMOVE(srcAddr := ADR(aiPimWorkStepHistoric[1]), destAddr := ADR(aiPimWorkStepHistoric[2]), n:= 9*SIZEOF(aiPimWorkStepHistoric[1]));
	aiPimWorkStepHistoric[1]:= iMemPimWorkStep;
END_IF
iMemPimWorkStep:=iWorkStep;

bOperationEnded:= FALSE;

bWorkPermitt := stPimInOut.bTestMode OR NOT stPimInOut.bPIMActive OR 
					(fbTON_UserLogedDeleyed.Q AND NOT stPimInOut.bWorkBlock_PIM AND NOT stPimInOut.bWorkBlock_PLC
					AND (NOT stPimInOut.bAlarmPLC OR stPimInOut.bNonBlockingAlarm)
					AND bMachineParamsOK AND bStationDataOK AND NOT bRetool AND NOT bMachParamsReadFromDB AND NOT bMachParamsSendToDB);
				
CASE iWorkStep OF
	-1: // PIM nieaktywny
		IF stPimInOut.bPIMActive THEN 
			stPimInOut.sPlcServiceMessage := '';
			iWorkStep := 0;
		END_IF
		
	0:		// Inicjalizacja stanowiska
		fbLogger.sDirectoryToSave:= CONCAT(STR1:= GVL_Aircom.sLogsPath, STR2:='PIM\');
		fbLogger.sFileNameWithFormat := CONCAT(STR1:= sStationName, STR2:=CONCAT(STR1:= '_M', STR2:=CONCAT(STR1:= INT_TO_STRING(iMachineNumber), STR2:= '.txt')));
		fbLogger(sNetId := '', sPreambule := GVL_Aircom.stAC_DT_Data.sTimeString,);
		stStationStatus.sLine := sLineName;
		stStationStatus.sStation := sStationName;
		stStationStatus.sNazwaStanowiska:= CONCAT(STR1:= CONCAT(STR1:= sStationName, '_'), INT_TO_STRING(iMachineNumber));
		stStationStatus.iMachineNumber := iMachineNumber;
		stStationStatus.bIsHidden := bIsHidden;
		stStationStatus.sNazwaStanowiska:= CONCAT(STR1:= CONCAT(STR1:= sStationName, '_'), INT_TO_STRING(iMachineNumber));
		bMachineParamsOK := bStationDataOK := bStationDataOK_Temp := FALSE;
		bSelectStationId := TRUE;	// Pobranie danych stanowiska z bazy danych
		iWorkStep := 5;
		
	5:	// Oczekiwanie na Pobranie danch stacji z bazy danych 
		IF NOT bSelectStationId THEN
			IF stRetDataLineStation.IdStacji <> 0 THEN	
				fbLogger.mAddLine(sTextToSave := CONCAT(STR1:= 'RecvStationId- ', STR2:= DINT_TO_STRING(stRetDataLineStation.IdStacji)));
				bStationDataOK := TRUE;
				iWorkStep := 10;
			ELSE
				mNewEvent(nInputErrorID := nPIM_ErrorCodes.SelectStationIdError, nEventType := nPIM_EventClasses.Error, tMessageTime := T#0S);
			END_IF
		END_IF

	10:	// Inicjalizacja zakończona OK, oczekiwanie na operacje z maszyny
		IF bRefreshData THEN
 			iWorkStep := 0;
			bRefreshData := FALSE;			
		ELSIF bSaveStatus THEN
			fbLogger.mAppendCurrentLine(bBreakLine := FALSE, sAddSep := '', sAppendText:= 'NewOperation');
			iCtr_Operations:= iCtr_Operations +1;
			bStatusToSaveMemory:= bStatusToSave;
			bStatusSavedOK := FALSE;
			iWorkStep := 15;
		END_IF
		
	15:	// Operacja trwa, oczekiwanie na zakończenie (możliwy pomiar czasu cyklu)
		IF bStatusToSave THEN
			iCtr_OperationsEndedOK:= iCtr_OperationsEndedOK +1;
			bOperationEnded:= bOperationStatus:= TRUE;
			m_SqlSelInsStatus(bStatus := TRUE, sErrCode := '', bSustein := TRUE);
			bStatusSaveTriggered := TRUE;
			bLockAfterStatusSave := FALSE;	
			iWorkStep := 20;
		ELSE
			iCtr_OperationsEndedNOK:= iCtr_OperationsEndedNOK +1;
			bOperationEnded:= TRUE;
			bOperationStatus:= FALSE;
			IF iEventId > 0 THEN
				mNewEvent(nEventType := nPIM_EventClasses.Error, nInputErrorID := iEventId, tMessageTime := T#0S);
			ELSE
				mNewEvent(nEventType := nPIM_EventClasses.Error, nInputErrorID := nPIM_ErrorCodes.UnKnownAlarm, tMessageTime := T#0S);
			END_IF
		END_IF
		iWorkStep := 20;
		
